(* CODESYS project mobject-graph-vision-pack.library
   Company: mobject
   Version: 0.7.0
   DefaultNamespace: mobject-graph-vision-pack
   Title: mobject-graph-vision-pack
   Placeholder: mobject-graph-vision-pack
   Author: mobject dev team
   DocFormat: reStructuredText

Project tree, tasks and I/O mapping:
  libraries: mobject-core, 0.5.0 (mobject); mobject-graph, 0.14.0 (mobject); mobject-graph-plc-pack, 0.15.0 (mobject); Tc2_Standard, * (Beckhoff Automation GmbH); Tc2_System, * (Beckhoff Automation GmbH); Tc3_Module, * (Beckhoff Automation GmbH); Tc3_Vision, * (Beckhoff Automation GmbH)
  Datatypes/
    Aliases/
      function block _GVCP_REGISTER_ADDRESS [ST]: SetBaseDatatypeReference, Address, ClearReference, Size, FB_init, Clone, Identifier, MakeReferenceTo, TryMakeReferenceTo, Value
      function block _TcVnArray10_ITcVnImage [ST]: SetBaseDatatypeReference, Address, ClearReference, Size, FB_init, Clone, Identifier, MakeReferenceTo, TryMakeReferenceTo, Value
      function block _TcVnArray3_Point2_REAL [ST]: SetBaseDatatypeReference, Address, ClearReference, Size, FB_init, Clone, Identifier, MakeReferenceTo, TryMakeReferenceTo, Value
      function block _TcVnArray4_LREAL [ST]: SetBaseDatatypeReference, Address, ClearReference, Size, FB_init, Clone, Identifier, MakeReferenceTo, TryMakeReferenceTo, Value
      function block _TcVnArray4_Point2_REAL [ST]: SetBaseDatatypeReference, Address, ClearReference, Size, FB_init, Clone, Identifier, MakeReferenceTo, TryMakeReferenceTo, Value
      function block _TcVnArray7_LREAL [ST]: SetBaseDatatypeReference, Address, ClearReference, Size, FB_init, Clone, Identifier, MakeReferenceTo, TryMakeReferenceTo, Value
      function block _TcVnArray8_LREAL [ST]: SetBaseDatatypeReference, Address, ClearReference, Size, FB_init, Clone, Identifier, MakeReferenceTo, TryMakeReferenceTo, Value
      function block _TcVnPoint [ST]: SetBaseDatatypeReference, Address, ClearReference, Size, FB_init, Clone, Identifier, MakeReferenceTo, TryMakeReferenceTo, Value
      function block _TcVnPoint2_DINT [ST]: SetBaseDatatypeReference, Address, ClearReference, Size, FB_init, Clone, Identifier, MakeReferenceTo, TryMakeReferenceTo, Value
      function block _TcVnPoint2_LREAL [ST]: SetBaseDatatypeReference, Address, ClearReference, Size, FB_init, Clone, Identifier, MakeReferenceTo, TryMakeReferenceTo, Value
      function block _TcVnPoint2_REAL [ST]: SetBaseDatatypeReference, Address, ClearReference, Size, FB_init, Clone, Identifier, MakeReferenceTo, TryMakeReferenceTo, Value
      function block _TcVnPoint3_LREAL [ST]: SetBaseDatatypeReference, Address, ClearReference, Size, FB_init, Clone, Identifier, MakeReferenceTo, TryMakeReferenceTo, Value
      function block _TcVnPoint3_REAL [ST]: SetBaseDatatypeReference, Address, ClearReference, Size, FB_init, Clone, Identifier, MakeReferenceTo, TryMakeReferenceTo, Value
      function block _TcVnRectangle [ST]: SetBaseDatatypeReference, Address, ClearReference, Size, FB_init, Clone, Identifier, MakeReferenceTo, TryMakeReferenceTo, Value
      function block _TcVnVector2_DINT [ST]: SetBaseDatatypeReference, Address, ClearReference, Size, FB_init, Clone, Identifier, MakeReferenceTo, TryMakeReferenceTo, Value
      function block _TcVnVector2_INT [ST]: SetBaseDatatypeReference, Address, ClearReference, Size, FB_init, Clone, Identifier, MakeReferenceTo, TryMakeReferenceTo, Value
      function block _TcVnVector2_LREAL [ST]: SetBaseDatatypeReference, Address, ClearReference, Size, FB_init, Clone, Identifier, MakeReferenceTo, TryMakeReferenceTo, Value
      function block _TcVnVector2_REAL [ST]: SetBaseDatatypeReference, Address, ClearReference, Size, FB_init, Clone, Identifier, MakeReferenceTo, TryMakeReferenceTo, Value
      function block _TcVnVector2_SINT [ST]: SetBaseDatatypeReference, Address, ClearReference, Size, FB_init, Clone, Identifier, MakeReferenceTo, TryMakeReferenceTo, Value
      function block _TcVnVector2_UINT [ST]: SetBaseDatatypeReference, Address, ClearReference, Size, FB_init, Clone, Identifier, MakeReferenceTo, TryMakeReferenceTo, Value
      function block _TcVnVector2_USINT [ST]: SetBaseDatatypeReference, Address, ClearReference, Size, FB_init, Clone, Identifier, MakeReferenceTo, TryMakeReferenceTo, Value
      function block _TcVnVector3_INT [ST]: SetBaseDatatypeReference, Address, ClearReference, Size, FB_init, Clone, Identifier, MakeReferenceTo, TryMakeReferenceTo, Value
      function block _TcVnVector3_LREAL [ST]: SetBaseDatatypeReference, Address, ClearReference, Size, FB_init, Clone, Identifier, MakeReferenceTo, TryMakeReferenceTo, Value
      function block _TcVnVector3_REAL [ST]: SetBaseDatatypeReference, Address, ClearReference, Size, FB_init, Clone, Identifier, MakeReferenceTo, TryMakeReferenceTo, Value
      function block _TcVnVector3_SINT [ST]: SetBaseDatatypeReference, Address, ClearReference, Size, FB_init, Clone, Identifier, MakeReferenceTo, TryMakeReferenceTo, Value
      function block _TcVnVector3_UINT [ST]: SetBaseDatatypeReference, Address, ClearReference, Size, FB_init, Clone, Identifier, MakeReferenceTo, TryMakeReferenceTo, Value
      function block _TcVnVector3_USINT [ST]: SetBaseDatatypeReference, Address, ClearReference, Size, FB_init, Clone, Identifier, MakeReferenceTo, TryMakeReferenceTo, Value
      function block _TcVnVector4_DINT [ST]: SetBaseDatatypeReference, Address, ClearReference, Size, FB_init, Clone, Identifier, MakeReferenceTo, TryMakeReferenceTo, Value
      function block _TcVnVector4_INT [ST]: SetBaseDatatypeReference, Address, ClearReference, Size, FB_init, Clone, Identifier, MakeReferenceTo, TryMakeReferenceTo, Value
      function block _TcVnVector4_LREAL [ST]: SetBaseDatatypeReference, Address, ClearReference, Size, FB_init, Clone, Identifier, MakeReferenceTo, TryMakeReferenceTo, Value
      function block _TcVnVector4_SINT [ST]: SetBaseDatatypeReference, Address, ClearReference, Size, FB_init, Clone, Identifier, MakeReferenceTo, TryMakeReferenceTo, Value
      function block _TcVnVector4_UINT [ST]: SetBaseDatatypeReference, Address, ClearReference, Size, FB_init, Clone, Identifier, MakeReferenceTo, TryMakeReferenceTo, Value
      function block _TcVnVector4_USINT [ST]: SetBaseDatatypeReference, Address, ClearReference, Size, FB_init, Clone, Identifier, MakeReferenceTo, TryMakeReferenceTo, Value
    Arrays/
      function block _Array0to1_0to2OfLREAL [ST]: FB_init, OnSerializeArrayValues, SetElementReference, TryDeserializeArrayValues, Address, BaseDatatype, ClearReference, Size, TryGetElementAsDatatypeByIndex, TryGetLowerBound, TryGetUpperBound, Clone, MakeReferenceTo, TryMakeReferenceTo, Value
      function block _Array0to1OfDINT [ST]: FB_init, OnSerializeArrayValues, SetElementReference, TryDeserializeArrayValues, Address, BaseDatatype, ClearReference, Size, TryGetElementAsDatatypeByIndex, TryGetLowerBound, TryGetUpperBound, Clone, MakeReferenceTo, TryMakeReferenceTo, Value
      function block _Array0to1OfINT [ST]: FB_init, OnSerializeArrayValues, SetElementReference, TryDeserializeArrayValues, Address, BaseDatatype, ClearReference, Size, TryGetElementAsDatatypeByIndex, TryGetLowerBound, TryGetUpperBound, Clone, MakeReferenceTo, TryMakeReferenceTo, Value
      function block _Array0to1OfLREAL [ST]: FB_init, OnSerializeArrayValues, SetElementReference, TryDeserializeArrayValues, Address, BaseDatatype, ClearReference, Size, TryGetElementAsDatatypeByIndex, TryGetLowerBound, TryGetUpperBound, Clone, MakeReferenceTo, TryMakeReferenceTo, Value
      function block _Array0to1OfREAL [ST]: FB_init, OnSerializeArrayValues, SetElementReference, TryDeserializeArrayValues, Address, BaseDatatype, ClearReference, Size, TryGetElementAsDatatypeByIndex, TryGetLowerBound, TryGetUpperBound, Clone, MakeReferenceTo, TryMakeReferenceTo, Value
      function block _Array0to1OfSINT [ST]: FB_init, OnSerializeArrayValues, SetElementReference, TryDeserializeArrayValues, Address, BaseDatatype, ClearReference, Size, TryGetElementAsDatatypeByIndex, TryGetLowerBound, TryGetUpperBound, Clone, MakeReferenceTo, TryMakeReferenceTo, Value
      function block _Array0to1OfUINT [ST]: FB_init, OnSerializeArrayValues, SetElementReference, TryDeserializeArrayValues, Address, BaseDatatype, ClearReference, Size, TryGetElementAsDatatypeByIndex, TryGetLowerBound, TryGetUpperBound, Clone, MakeReferenceTo, TryMakeReferenceTo, Value
      function block _Array0to1OfUSINT [ST]: FB_init, OnSerializeArrayValues, SetElementReference, TryDeserializeArrayValues, Address, BaseDatatype, ClearReference, Size, TryGetElementAsDatatypeByIndex, TryGetLowerBound, TryGetUpperBound, Clone, MakeReferenceTo, TryMakeReferenceTo, Value
      function block _Array0to2_0to2OfLREAL [ST]: FB_init, OnSerializeArrayValues, SetElementReference, TryDeserializeArrayValues, Address, BaseDatatype, ClearReference, Size, TryGetElementAsDatatypeByIndex, TryGetLowerBound, TryGetUpperBound, Clone, MakeReferenceTo, TryMakeReferenceTo, Value
      function block _Array0to2OfINT [ST]: FB_init, OnSerializeArrayValues, SetElementReference, TryDeserializeArrayValues, Address, BaseDatatype, ClearReference, Size, TryGetElementAsDatatypeByIndex, TryGetLowerBound, TryGetUpperBound, Clone, MakeReferenceTo, TryMakeReferenceTo, Value
      function block _Array0to2OfLREAL [ST]: FB_init, OnSerializeArrayValues, SetElementReference, TryDeserializeArrayValues, Address, BaseDatatype, ClearReference, Size, TryGetElementAsDatatypeByIndex, TryGetLowerBound, TryGetUpperBound, Clone, MakeReferenceTo, TryMakeReferenceTo, Value
      function block _Array0to2OfREAL [ST]: FB_init, OnSerializeArrayValues, SetElementReference, TryDeserializeArrayValues, Address, BaseDatatype, ClearReference, Size, TryGetElementAsDatatypeByIndex, TryGetLowerBound, TryGetUpperBound, Clone, MakeReferenceTo, TryMakeReferenceTo, Value
      function block _Array0to2OfSINT [ST]: FB_init, OnSerializeArrayValues, SetElementReference, TryDeserializeArrayValues, Address, BaseDatatype, ClearReference, Size, TryGetElementAsDatatypeByIndex, TryGetLowerBound, TryGetUpperBound, Clone, MakeReferenceTo, TryMakeReferenceTo, Value
      function block _Array0to2OfTcVnPoint2_REAL [ST]: FB_init, OnSerializeArrayValues, SetElementReference, TryDeserializeArrayValues, Address, BaseDatatype, ClearReference, Size, TryGetElementAsDatatypeByIndex, TryGetLowerBound, TryGetUpperBound, Clone, MakeReferenceTo, TryMakeReferenceTo, Value
      function block _Array0to2OfUINT [ST]: FB_init, OnSerializeArrayValues, SetElementReference, TryDeserializeArrayValues, Address, BaseDatatype, ClearReference, Size, TryGetElementAsDatatypeByIndex, TryGetLowerBound, TryGetUpperBound, Clone, MakeReferenceTo, TryMakeReferenceTo, Value
      function block _Array0to2OfUSINT [ST]: FB_init, OnSerializeArrayValues, SetElementReference, TryDeserializeArrayValues, Address, BaseDatatype, ClearReference, Size, TryGetElementAsDatatypeByIndex, TryGetLowerBound, TryGetUpperBound, Clone, MakeReferenceTo, TryMakeReferenceTo, Value
      function block _Array0to32OfUDINT [ST]: FB_init, OnSerializeArrayValues, SetElementReference, TryDeserializeArrayValues, Address, BaseDatatype, ClearReference, Size, TryGetElementAsDatatypeByIndex, TryGetLowerBound, TryGetUpperBound, Clone, MakeReferenceTo, TryMakeReferenceTo, Value
      function block _Array0to3OfDINT [ST]: FB_init, OnSerializeArrayValues, SetElementReference, TryDeserializeArrayValues, Address, BaseDatatype, ClearReference, Size, TryGetElementAsDatatypeByIndex, TryGetLowerBound, TryGetUpperBound, Clone, MakeReferenceTo, TryMakeReferenceTo, Value
      function block _Array0to3OfINT [ST]: FB_init, OnSerializeArrayValues, SetElementReference, TryDeserializeArrayValues, Address, BaseDatatype, ClearReference, Size, TryGetElementAsDatatypeByIndex, TryGetLowerBound, TryGetUpperBound, Clone, MakeReferenceTo, TryMakeReferenceTo, Value
      function block _Array0to3OfLREAL [ST]: FB_init, OnSerializeArrayValues, SetElementReference, TryDeserializeArrayValues, Address, BaseDatatype, ClearReference, Size, TryGetElementAsDatatypeByIndex, TryGetLowerBound, TryGetUpperBound, Clone, MakeReferenceTo, TryMakeReferenceTo, Value
      function block _Array0to3OfSINT [ST]: FB_init, OnSerializeArrayValues, SetElementReference, TryDeserializeArrayValues, Address, BaseDatatype, ClearReference, Size, TryGetElementAsDatatypeByIndex, TryGetLowerBound, TryGetUpperBound, Clone, MakeReferenceTo, TryMakeReferenceTo, Value
      function block _Array0to3OfTcVnPoint2_REAL [ST]: FB_init, OnSerializeArrayValues, SetElementReference, TryDeserializeArrayValues, Address, BaseDatatype, ClearReference, Size, TryGetElementAsDatatypeByIndex, TryGetLowerBound, TryGetUpperBound, Clone, MakeReferenceTo, TryMakeReferenceTo, Value
      function block _Array0to3OfUINT [ST]: FB_init, OnSerializeArrayValues, SetElementReference, TryDeserializeArrayValues, Address, BaseDatatype, ClearReference, Size, TryGetElementAsDatatypeByIndex, TryGetLowerBound, TryGetUpperBound, Clone, MakeReferenceTo, TryMakeReferenceTo, Value
      function block _Array0to3OfUSINT [ST]: FB_init, OnSerializeArrayValues, SetElementReference, TryDeserializeArrayValues, Address, BaseDatatype, ClearReference, Size, TryGetElementAsDatatypeByIndex, TryGetLowerBound, TryGetUpperBound, Clone, MakeReferenceTo, TryMakeReferenceTo, Value
      function block _Array0to6OfLREAL [ST]: FB_init, OnSerializeArrayValues, SetElementReference, TryDeserializeArrayValues, Address, BaseDatatype, ClearReference, Size, TryGetElementAsDatatypeByIndex, TryGetLowerBound, TryGetUpperBound, Clone, MakeReferenceTo, TryMakeReferenceTo, Value
      function block _Array0to7OfLREAL [ST]: FB_init, OnSerializeArrayValues, SetElementReference, TryDeserializeArrayValues, Address, BaseDatatype, ClearReference, Size, TryGetElementAsDatatypeByIndex, TryGetLowerBound, TryGetUpperBound, Clone, MakeReferenceTo, TryMakeReferenceTo, Value
      function block _Array0to9OfITcVnImage [ST]: FB_init, OnSerializeArrayValues, SetElementReference, TryDeserializeArrayValues, Address, BaseDatatype, ClearReference, Size, TryGetElementAsDatatypeByIndex, TryGetLowerBound, TryGetUpperBound, Clone, MakeReferenceTo, TryMakeReferenceTo, Value
    Enums/
      function block _ETcVn2dCodeSearchStrategy [ST]: SetBaseDatatypeReference, Address, ClearReference, Size, FB_init, AddLocalEnumeration, IsEnumeratorValueEqual, Clone, Identifier, MakeReferenceTo, TryMakeReferenceTo, Value
      function block _ETcVnAdaptiveThresholdMethod [ST]: SetBaseDatatypeReference, Address, ClearReference, Size, FB_init, AddLocalEnumeration, IsEnumeratorValueEqual, Clone, Identifier, MakeReferenceTo, TryMakeReferenceTo, Value
      function block _ETcVnBarcodeSearchDirection [ST]: SetBaseDatatypeReference, Address, ClearReference, Size, FB_init, AddLocalEnumeration, IsEnumeratorValueEqual, Clone, Identifier, MakeReferenceTo, TryMakeReferenceTo, Value
      function block _ETcVnBarcodeType [ST]: SetBaseDatatypeReference, Address, ClearReference, Size, FB_init, AddLocalEnumeration, IsEnumeratorValueEqual, Clone, Identifier, MakeReferenceTo, TryMakeReferenceTo, Value
      function block _ETcVnBlobCombination [ST]: SetBaseDatatypeReference, Address, ClearReference, Size, FB_init, AddLocalEnumeration, IsEnumeratorValueEqual, Clone, Identifier, MakeReferenceTo, TryMakeReferenceTo, Value
      function block _ETcVnBorderInterpolationMethod [ST]: SetBaseDatatypeReference, Address, ClearReference, Size, FB_init, AddLocalEnumeration, IsEnumeratorValueEqual, Clone, Identifier, MakeReferenceTo, TryMakeReferenceTo, Value
      function block _ETcVnCalibrationPattern [ST]: SetBaseDatatypeReference, Address, ClearReference, Size, FB_init, AddLocalEnumeration, IsEnumeratorValueEqual, Clone, Identifier, MakeReferenceTo, TryMakeReferenceTo, Value
      function block _ETcVnCalibrationPatternOrigin [ST]: SetBaseDatatypeReference, Address, ClearReference, Size, FB_init, AddLocalEnumeration, IsEnumeratorValueEqual, Clone, Identifier, MakeReferenceTo, TryMakeReferenceTo, Value
      function block _ETcVnCameraState [ST]: SetBaseDatatypeReference, Address, ClearReference, Size, FB_init, AddLocalEnumeration, IsEnumeratorValueEqual, Clone, Identifier, MakeReferenceTo, TryMakeReferenceTo, Value
      function block _ETcVnClusteringAlgorithm [ST]: SetBaseDatatypeReference, Address, ClearReference, Size, FB_init, AddLocalEnumeration, IsEnumeratorValueEqual, Clone, Identifier, MakeReferenceTo, TryMakeReferenceTo, Value
      function block _ETcVnColorMap [ST]: SetBaseDatatypeReference, Address, ClearReference, Size, FB_init, AddLocalEnumeration, IsEnumeratorValueEqual, Clone, Identifier, MakeReferenceTo, TryMakeReferenceTo, Value
      function block _ETcVnColorMapSize [ST]: SetBaseDatatypeReference, Address, ClearReference, Size, FB_init, AddLocalEnumeration, IsEnumeratorValueEqual, Clone, Identifier, MakeReferenceTo, TryMakeReferenceTo, Value
      function block _ETcVnColorSpaceTransform [ST]: SetBaseDatatypeReference, Address, ClearReference, Size, FB_init, AddLocalEnumeration, IsEnumeratorValueEqual, Clone, Identifier, MakeReferenceTo, TryMakeReferenceTo, Value
      function block _ETcVnColorTrainingMethod [ST]: SetBaseDatatypeReference, Address, ClearReference, Size, FB_init, AddLocalEnumeration, IsEnumeratorValueEqual, Clone, Identifier, MakeReferenceTo, TryMakeReferenceTo, Value
      function block _ETcVnConnectedComponentsAlgorithm [ST]: SetBaseDatatypeReference, Address, ClearReference, Size, FB_init, AddLocalEnumeration, IsEnumeratorValueEqual, Clone, Identifier, MakeReferenceTo, TryMakeReferenceTo, Value
      function block _ETcVnContainerExportFormat [ST]: SetBaseDatatypeReference, Address, ClearReference, Size, FB_init, AddLocalEnumeration, IsEnumeratorValueEqual, Clone, Identifier, MakeReferenceTo, TryMakeReferenceTo, Value
      function block _ETcVnContourApproximationMethod [ST]: SetBaseDatatypeReference, Address, ClearReference, Size, FB_init, AddLocalEnumeration, IsEnumeratorValueEqual, Clone, Identifier, MakeReferenceTo, TryMakeReferenceTo, Value
      function block _ETcVnContourRetrievalMode [ST]: SetBaseDatatypeReference, Address, ClearReference, Size, FB_init, AddLocalEnumeration, IsEnumeratorValueEqual, Clone, Identifier, MakeReferenceTo, TryMakeReferenceTo, Value
      function block _ETcVnContoursMatchComparisonMethod [ST]: SetBaseDatatypeReference, Address, ClearReference, Size, FB_init, AddLocalEnumeration, IsEnumeratorValueEqual, Clone, Identifier, MakeReferenceTo, TryMakeReferenceTo, Value
      function block _ETcVnDiffusivityTypeKAZE [ST]: SetBaseDatatypeReference, Address, ClearReference, Size, FB_init, AddLocalEnumeration, IsEnumeratorValueEqual, Clone, Identifier, MakeReferenceTo, TryMakeReferenceTo, Value
      function block _ETcVnDistanceTransformationLabel [ST]: SetBaseDatatypeReference, Address, ClearReference, Size, FB_init, AddLocalEnumeration, IsEnumeratorValueEqual, Clone, Identifier, MakeReferenceTo, TryMakeReferenceTo, Value
      function block _ETcVnDistanceTransformationMask [ST]: SetBaseDatatypeReference, Address, ClearReference, Size, FB_init, AddLocalEnumeration, IsEnumeratorValueEqual, Clone, Identifier, MakeReferenceTo, TryMakeReferenceTo, Value
      function block _ETcVnDistanceType [ST]: SetBaseDatatypeReference, Address, ClearReference, Size, FB_init, AddLocalEnumeration, IsEnumeratorValueEqual, Clone, Identifier, MakeReferenceTo, TryMakeReferenceTo, Value
      function block _ETcVnDrawMatchesFlags [ST]: SetBaseDatatypeReference, Address, ClearReference, Size, FB_init, AddLocalEnumeration, IsEnumeratorValueEqual, Clone, Identifier, MakeReferenceTo, TryMakeReferenceTo, Value
      function block _ETcVnDrawShape [ST]: SetBaseDatatypeReference, Address, ClearReference, Size, FB_init, AddLocalEnumeration, IsEnumeratorValueEqual, Clone, Identifier, MakeReferenceTo, TryMakeReferenceTo, Value
      function block _ETcVnEdgeDetectionAlgorithm [ST]: SetBaseDatatypeReference, Address, ClearReference, Size, FB_init, AddLocalEnumeration, IsEnumeratorValueEqual, Clone, Identifier, MakeReferenceTo, TryMakeReferenceTo, Value
      function block _ETcVnEdgeDirection [ST]: SetBaseDatatypeReference, Address, ClearReference, Size, FB_init, AddLocalEnumeration, IsEnumeratorValueEqual, Clone, Identifier, MakeReferenceTo, TryMakeReferenceTo, Value
      function block _ETcVnElementType [ST]: SetBaseDatatypeReference, Address, ClearReference, Size, FB_init, AddLocalEnumeration, IsEnumeratorValueEqual, Clone, Identifier, MakeReferenceTo, TryMakeReferenceTo, Value
      function block _ETcVnEstimationAlgorithm [ST]: SetBaseDatatypeReference, Address, ClearReference, Size, FB_init, AddLocalEnumeration, IsEnumeratorValueEqual, Clone, Identifier, MakeReferenceTo, TryMakeReferenceTo, Value
      function block _ETcVnExtremePointDirection [ST]: SetBaseDatatypeReference, Address, ClearReference, Size, FB_init, AddLocalEnumeration, IsEnumeratorValueEqual, Clone, Identifier, MakeReferenceTo, TryMakeReferenceTo, Value
      function block _ETcVnFeatureDescriptorTypeAKAZE [ST]: SetBaseDatatypeReference, Address, ClearReference, Size, FB_init, AddLocalEnumeration, IsEnumeratorValueEqual, Clone, Identifier, MakeReferenceTo, TryMakeReferenceTo, Value
      function block _ETcVnFeatureScoreTypeORB [ST]: SetBaseDatatypeReference, Address, ClearReference, Size, FB_init, AddLocalEnumeration, IsEnumeratorValueEqual, Clone, Identifier, MakeReferenceTo, TryMakeReferenceTo, Value
      function block _ETcVnFilterDirection [ST]: SetBaseDatatypeReference, Address, ClearReference, Size, FB_init, AddLocalEnumeration, IsEnumeratorValueEqual, Clone, Identifier, MakeReferenceTo, TryMakeReferenceTo, Value
      function block _ETcVnFlipAxis [ST]: SetBaseDatatypeReference, Address, ClearReference, Size, FB_init, AddLocalEnumeration, IsEnumeratorValueEqual, Clone, Identifier, MakeReferenceTo, TryMakeReferenceTo, Value
      function block _ETcVnFontType [ST]: SetBaseDatatypeReference, Address, ClearReference, Size, FB_init, AddLocalEnumeration, IsEnumeratorValueEqual, Clone, Identifier, MakeReferenceTo, TryMakeReferenceTo, Value
      function block _ETcVnHoughMethod [ST]: SetBaseDatatypeReference, Address, ClearReference, Size, FB_init, AddLocalEnumeration, IsEnumeratorValueEqual, Clone, Identifier, MakeReferenceTo, TryMakeReferenceTo, Value
      function block _ETcVnInterpolationType [ST]: SetBaseDatatypeReference, Address, ClearReference, Size, FB_init, AddLocalEnumeration, IsEnumeratorValueEqual, Clone, Identifier, MakeReferenceTo, TryMakeReferenceTo, Value
      function block _ETcVnKeypointDetectionTypeAGAST [ST]: SetBaseDatatypeReference, Address, ClearReference, Size, FB_init, AddLocalEnumeration, IsEnumeratorValueEqual, Clone, Identifier, MakeReferenceTo, TryMakeReferenceTo, Value
      function block _ETcVnKeypointDetectionTypeFAST [ST]: SetBaseDatatypeReference, Address, ClearReference, Size, FB_init, AddLocalEnumeration, IsEnumeratorValueEqual, Clone, Identifier, MakeReferenceTo, TryMakeReferenceTo, Value
      function block _ETcVnLineType [ST]: SetBaseDatatypeReference, Address, ClearReference, Size, FB_init, AddLocalEnumeration, IsEnumeratorValueEqual, Clone, Identifier, MakeReferenceTo, TryMakeReferenceTo, Value
      function block _ETcVnMorphologicalOperator [ST]: SetBaseDatatypeReference, Address, ClearReference, Size, FB_init, AddLocalEnumeration, IsEnumeratorValueEqual, Clone, Identifier, MakeReferenceTo, TryMakeReferenceTo, Value
      function block _ETcVnNormalizationType [ST]: SetBaseDatatypeReference, Address, ClearReference, Size, FB_init, AddLocalEnumeration, IsEnumeratorValueEqual, Clone, Identifier, MakeReferenceTo, TryMakeReferenceTo, Value
      function block _ETcVnOrientationMethod [ST]: SetBaseDatatypeReference, Address, ClearReference, Size, FB_init, AddLocalEnumeration, IsEnumeratorValueEqual, Clone, Identifier, MakeReferenceTo, TryMakeReferenceTo, Value
      function block _ETcVnPixelConnectivity [ST]: SetBaseDatatypeReference, Address, ClearReference, Size, FB_init, AddLocalEnumeration, IsEnumeratorValueEqual, Clone, Identifier, MakeReferenceTo, TryMakeReferenceTo, Value
      function block _ETcVnPixelEncoding [ST]: SetBaseDatatypeReference, Address, ClearReference, Size, FB_init, AddLocalEnumeration, IsEnumeratorValueEqual, Clone, Identifier, MakeReferenceTo, TryMakeReferenceTo, Value
      function block _ETcVnPixelPackMode [ST]: SetBaseDatatypeReference, Address, ClearReference, Size, FB_init, AddLocalEnumeration, IsEnumeratorValueEqual, Clone, Identifier, MakeReferenceTo, TryMakeReferenceTo, Value
      function block _ETcVnRectangleIntersection [ST]: SetBaseDatatypeReference, Address, ClearReference, Size, FB_init, AddLocalEnumeration, IsEnumeratorValueEqual, Clone, Identifier, MakeReferenceTo, TryMakeReferenceTo, Value
      function block _ETcVnRotationAngle [ST]: SetBaseDatatypeReference, Address, ClearReference, Size, FB_init, AddLocalEnumeration, IsEnumeratorValueEqual, Clone, Identifier, MakeReferenceTo, TryMakeReferenceTo, Value
      function block _ETcVnSignedNormalization [ST]: SetBaseDatatypeReference, Address, ClearReference, Size, FB_init, AddLocalEnumeration, IsEnumeratorValueEqual, Clone, Identifier, MakeReferenceTo, TryMakeReferenceTo, Value
      function block _ETcVnStructuringElementShape [ST]: SetBaseDatatypeReference, Address, ClearReference, Size, FB_init, AddLocalEnumeration, IsEnumeratorValueEqual, Clone, Identifier, MakeReferenceTo, TryMakeReferenceTo, Value
      function block _ETcVnTemplateMatchMethod [ST]: SetBaseDatatypeReference, Address, ClearReference, Size, FB_init, AddLocalEnumeration, IsEnumeratorValueEqual, Clone, Identifier, MakeReferenceTo, TryMakeReferenceTo, Value
      function block _ETcVnThresholdType [ST]: SetBaseDatatypeReference, Address, ClearReference, Size, FB_init, AddLocalEnumeration, IsEnumeratorValueEqual, Clone, Identifier, MakeReferenceTo, TryMakeReferenceTo, Value
      function block _ETcVnVectorCompareMethod [ST]: SetBaseDatatypeReference, Address, ClearReference, Size, FB_init, AddLocalEnumeration, IsEnumeratorValueEqual, Clone, Identifier, MakeReferenceTo, TryMakeReferenceTo, Value
      function block _ETcVnWorldCoordinateSystem [ST]: SetBaseDatatypeReference, Address, ClearReference, Size, FB_init, AddLocalEnumeration, IsEnumeratorValueEqual, Clone, Identifier, MakeReferenceTo, TryMakeReferenceTo, Value
      function block _ETcWatchdogAccumulationType [ST]: SetBaseDatatypeReference, Address, ClearReference, Size, FB_init, AddLocalEnumeration, IsEnumeratorValueEqual, Clone, Identifier, MakeReferenceTo, TryMakeReferenceTo, Value
      function block _GEV_CAMERA_STATE [ST]: SetBaseDatatypeReference, Address, ClearReference, Size, FB_init, AddLocalEnumeration, IsEnumeratorValueEqual, Clone, Identifier, MakeReferenceTo, TryMakeReferenceTo, Value
    Interfaces/
      function block _ITcVnContainer [ST]: Address, ClearReference, Size, FB_exit, Serialize_ContainerType_Vector_DINT, Serialize_ContainerType_Vector_INT, Serialize_ContainerType_Vector_ITcVnImage, Serialize_ContainerType_Vector_LREAL, Serialize_ContainerType_Vector_REAL, Serialize_ContainerType_Vector_SINT, Serialize_ContainerType_Vector_UDINT, Serialize_ContainerType_Vector_UINT, Serialize_ContainerType_Vector_ULINT, Serialize_ContainerType_Vector_USINT, TryTcReleaseLocal, Clone, Identifier, MakeReferenceTo, SerializeWith, TryDeserializeFrom, TryMakeReferenceTo, Value, HasType, IsValid, TryGetTypeName, TryTcAddRef, TryTcRelease
      function block _ITcVnImage [ST]: Address, ClearReference, Size, FB_exit, TryGetElementTypeFromInfo, TryTcReleaseLocal, Clone, Identifier, MakeReferenceTo, SerializeWith, TryMakeReferenceTo, Value, HasChannelCount, IsPixelValueCompatible, IsValid, TryDeserializeFrom, TryGetHeight, TryGetImageData, TryGetImageInfo, TryGetImageSize, TryGetPixelFormat, TryGetRowPointer, TryGetWidth, TryGetXPadding, TryGetYPadding, TryReleaseRowPointer, TryTcAddRef, TryTcRelease
    Structs/
      function block _TcVnCircularArc [ST]: Address, ClearReference, Size, FB_init, SetMemberReference, Clone, Identifier, MakeReferenceTo, TryMakeReferenceTo, Value, aCenter, fEndAngle, fRadius, fStartAngle
      function block _TcVnDMatch [ST]: Address, ClearReference, Size, FB_init, SetMemberReference, Clone, Identifier, MakeReferenceTo, TryMakeReferenceTo, Value, fDistance, nImageIdx, nQueryIdx, nTrainIdx
      function block _TcVnImageInfo [ST]: Address, ClearReference, Size, FB_init, SetMemberReference, Clone, Identifier, MakeReferenceTo, TryMakeReferenceTo, Value, nHeight, nImageSize, nWidth, nXPadding, nYPadding, stPixelFormat
      function block _TcVnKeyPoint [ST]: Address, ClearReference, Size, FB_init, SetMemberReference, Clone, Identifier, MakeReferenceTo, TryMakeReferenceTo, Value, aPoint, fAngle, fDiameter, fResponse, nClassId, nOctave
      function block _TcVnParamsBlobDetection [ST]: Address, ClearReference, Size, FB_init, SetMemberReference, Clone, Identifier, MakeReferenceTo, TryMakeReferenceTo, Value, bFilterByArea, bFilterByCircularity, bFilterByConvexity, bFilterByEccentricity, bFilterByInertiaRatio, eBlobCombination, eThresholdType, fMaxArea, fMaxCircularity, fMaxConvexity, fMaxEccentricity, fMaxInertiaRatio, fMaxThreshold, fMinArea, fMinBlobDistance, fMinCircularity, fMinConvexity, fMinEccentricity, fMinInertiaRatio, fMinThreshold, fThresholdStep, nMinRepeatability
      function block _TcVnPixelFormat [ST]: Address, ClearReference, Size, FB_init, SetMemberReference, Clone, Identifier, MakeReferenceTo, TryMakeReferenceTo, Value, bFloat, bPlanar, bSigned, bSupported, ePixelEncoding, ePixelPackMode, nChannels, nElementSize, nTotalSize
      function block _TcVnRectangle_DINT [ST]: Address, ClearReference, Size, FB_init, SetMemberReference, Clone, Identifier, MakeReferenceTo, TryMakeReferenceTo, Value, nHeight, nWidth, nX, nY
      function block _TcVnRectangle_UDINT [ST]: Address, ClearReference, Size, FB_init, SetMemberReference, Clone, Identifier, MakeReferenceTo, TryMakeReferenceTo, Value, nHeight, nWidth, nX, nY
      function block _TcVnRotatedRectangle [ST]: Address, ClearReference, Size, FB_init, SetMemberReference, Clone, Identifier, MakeReferenceTo, TryMakeReferenceTo, Value, aCenter, fAngle, stSize
      function block _TcVnSize2_REAL [ST]: Address, ClearReference, Size, FB_init, SetMemberReference, Clone, Identifier, MakeReferenceTo, TryMakeReferenceTo, Value, fHeight, fWidth
    function block VisionDatatypePack [ST]: RegisterWithDatatypes
  Nodes/
    Algebraic Container Operations/
    Algebraic Image Operations/
      function block Node_F_VN_BitwiseAndImages [ST]: FB_init, Clone, OnExecute, PreExecutionCheck
      function block Node_F_VN_BitwiseNotImage [ST]: FB_init, Clone, OnExecute, PreExecutionCheck
      function block Node_F_VN_BitwiseOrImages [ST]: FB_init, Clone, OnExecute, PreExecutionCheck
      function block Node_F_VN_BitwiseXorImages [ST]: FB_init, Clone, OnExecute, PreExecutionCheck
    Basic Container Operations/
      function block Node_F_VN_AppendToContainer_DINT [ST]: FB_init, Clone, OnExecute, PreExecutionCheck
      function block Node_F_VN_AppendToContainer_INT [ST]: FB_init, Clone, OnExecute, PreExecutionCheck
      function block Node_F_VN_AppendToContainer_ITcVnContainer [ST]: FB_init, Clone, OnExecute, PreExecutionCheck
      function block Node_F_VN_AppendToContainer_ITcVnImage [ST]: FB_init, Clone, OnExecute, PreExecutionCheck
      function block Node_F_VN_AppendToContainer_LREAL [ST]: FB_init, Clone, OnExecute, PreExecutionCheck
      function block Node_F_VN_AppendToContainer_REAL [ST]: FB_init, Clone, OnExecute, PreExecutionCheck
      function block Node_F_VN_AppendToContainer_SINT [ST]: FB_init, Clone, OnExecute, PreExecutionCheck
      function block Node_F_VN_AppendToContainer_TcVnDMatch [ST]: FB_init, Clone, OnExecute, PreExecutionCheck
      function block Node_F_VN_AppendToContainer_TcVnKeyPoint [ST]: FB_init, Clone, OnExecute, PreExecutionCheck
      function block Node_F_VN_AppendToContainer_TcVnPoint2_DINT [ST]: FB_init, Clone, OnExecute, PreExecutionCheck
      function block Node_F_VN_AppendToContainer_TcVnPoint2_LREAL [ST]: FB_init, Clone, OnExecute, PreExecutionCheck
      function block Node_F_VN_AppendToContainer_TcVnPoint2_REAL [ST]: FB_init, Clone, OnExecute, PreExecutionCheck
      function block Node_F_VN_AppendToContainer_TcVnPoint3_LREAL [ST]: FB_init, Clone, OnExecute, PreExecutionCheck
      function block Node_F_VN_AppendToContainer_TcVnPoint3_REAL [ST]: FB_init, Clone, OnExecute, PreExecutionCheck
      function block Node_F_VN_AppendToContainer_TcVnRectangle_DINT [ST]: FB_init, Clone, OnExecute, PreExecutionCheck
      function block Node_F_VN_AppendToContainer_TcVnVector2_DINT [ST]: FB_init, Clone, OnExecute, PreExecutionCheck
      function block Node_F_VN_AppendToContainer_TcVnVector2_INT [ST]: FB_init, Clone, OnExecute, PreExecutionCheck
      function block Node_F_VN_AppendToContainer_TcVnVector2_REAL [ST]: FB_init, Clone, OnExecute, PreExecutionCheck
      function block Node_F_VN_AppendToContainer_TcVnVector2_SINT [ST]: FB_init, Clone, OnExecute, PreExecutionCheck
      function block Node_F_VN_AppendToContainer_TcVnVector2_UINT [ST]: FB_init, Clone, OnExecute, PreExecutionCheck
      function block Node_F_VN_AppendToContainer_TcVnVector2_USINT [ST]: FB_init, Clone, OnExecute, PreExecutionCheck
      function block Node_F_VN_AppendToContainer_TcVnVector3_INT [ST]: FB_init, Clone, OnExecute, PreExecutionCheck
      function block Node_F_VN_AppendToContainer_TcVnVector3_REAL [ST]: FB_init, Clone, OnExecute, PreExecutionCheck
      function block Node_F_VN_AppendToContainer_TcVnVector3_SINT [ST]: FB_init, Clone, OnExecute, PreExecutionCheck
      function block Node_F_VN_AppendToContainer_TcVnVector3_UINT [ST]: FB_init, Clone, OnExecute, PreExecutionCheck
      function block Node_F_VN_AppendToContainer_TcVnVector3_USINT [ST]: FB_init, Clone, OnExecute, PreExecutionCheck
      function block Node_F_VN_AppendToContainer_TcVnVector4_DINT [ST]: FB_init, Clone, OnExecute, PreExecutionCheck
      function block Node_F_VN_AppendToContainer_TcVnVector4_INT [ST]: FB_init, Clone, OnExecute, PreExecutionCheck
      function block Node_F_VN_AppendToContainer_TcVnVector4_LREAL [ST]: FB_init, Clone, OnExecute, PreExecutionCheck
      function block Node_F_VN_AppendToContainer_TcVnVector4_SINT [ST]: FB_init, Clone, OnExecute, PreExecutionCheck
      function block Node_F_VN_AppendToContainer_TcVnVector4_UINT [ST]: FB_init, Clone, OnExecute, PreExecutionCheck
      function block Node_F_VN_AppendToContainer_TcVnVector4_USINT [ST]: FB_init, Clone, OnExecute, PreExecutionCheck
      function block Node_F_VN_AppendToContainer_UDINT [ST]: FB_init, Clone, OnExecute, PreExecutionCheck
      function block Node_F_VN_AppendToContainer_UINT [ST]: FB_init, Clone, OnExecute, PreExecutionCheck
      function block Node_F_VN_AppendToContainer_ULINT [ST]: FB_init, Clone, OnExecute, PreExecutionCheck
      function block Node_F_VN_AppendToContainer_USINT [ST]: FB_init, Clone, OnExecute, PreExecutionCheck
      function block Node_F_VN_FillContainer_DINT [ST]: FB_init, Clone, OnExecute, PreExecutionCheck
      function block Node_F_VN_FillContainer_INT [ST]: FB_init, Clone, OnExecute, PreExecutionCheck
      function block Node_F_VN_FillContainer_ITcVnImage [ST]: FB_init, Clone, OnExecute, PreExecutionCheck
      function block Node_F_VN_FillContainer_LREAL [ST]: FB_init, Clone, OnExecute, PreExecutionCheck
      function block Node_F_VN_FillContainer_REAL [ST]: FB_init, Clone, OnExecute, PreExecutionCheck
      function block Node_F_VN_FillContainer_SINT [ST]: FB_init, Clone, OnExecute, PreExecutionCheck
      function block Node_F_VN_FillContainer_TcVnDMatch [ST]: FB_init, Clone, OnExecute, PreExecutionCheck
      function block Node_F_VN_FillContainer_TcVnKeyPoint [ST]: FB_init, Clone, OnExecute, PreExecutionCheck
      function block Node_F_VN_FillContainer_TcVnPoint2_DINT [ST]: FB_init, Clone, OnExecute, PreExecutionCheck
      function block Node_F_VN_FillContainer_TcVnPoint2_LREAL [ST]: FB_init, Clone, OnExecute, PreExecutionCheck
      function block Node_F_VN_FillContainer_TcVnPoint2_REAL [ST]: FB_init, Clone, OnExecute, PreExecutionCheck
      function block Node_F_VN_FillContainer_TcVnPoint3_LREAL [ST]: FB_init, Clone, OnExecute, PreExecutionCheck
      function block Node_F_VN_FillContainer_TcVnPoint3_REAL [ST]: FB_init, Clone, OnExecute, PreExecutionCheck
      function block Node_F_VN_FillContainer_TcVnRectangle_DINT [ST]: FB_init, Clone, OnExecute, PreExecutionCheck
      function block Node_F_VN_FillContainer_TcVnVector2_DINT [ST]: FB_init, Clone, OnExecute, PreExecutionCheck
      function block Node_F_VN_FillContainer_TcVnVector2_INT [ST]: FB_init, Clone, OnExecute, PreExecutionCheck
      function block Node_F_VN_FillContainer_TcVnVector2_REAL [ST]: FB_init, Clone, OnExecute, PreExecutionCheck
      function block Node_F_VN_FillContainer_TcVnVector2_SINT [ST]: FB_init, Clone, OnExecute, PreExecutionCheck
      function block Node_F_VN_FillContainer_TcVnVector2_UINT [ST]: FB_init, Clone, OnExecute, PreExecutionCheck
      function block Node_F_VN_FillContainer_TcVnVector2_USINT [ST]: FB_init, Clone, OnExecute, PreExecutionCheck
      function block Node_F_VN_FillContainer_TcVnVector3_INT [ST]: FB_init, Clone, OnExecute, PreExecutionCheck
      function block Node_F_VN_FillContainer_TcVnVector3_REAL [ST]: FB_init, Clone, OnExecute, PreExecutionCheck
      function block Node_F_VN_FillContainer_TcVnVector3_SINT [ST]: FB_init, Clone, OnExecute, PreExecutionCheck
      function block Node_F_VN_FillContainer_TcVnVector3_UINT [ST]: FB_init, Clone, OnExecute, PreExecutionCheck
      function block Node_F_VN_FillContainer_TcVnVector3_USINT [ST]: FB_init, Clone, OnExecute, PreExecutionCheck
      function block Node_F_VN_FillContainer_TcVnVector4_DINT [ST]: FB_init, Clone, OnExecute, PreExecutionCheck
      function block Node_F_VN_FillContainer_TcVnVector4_INT [ST]: FB_init, Clone, OnExecute, PreExecutionCheck
      function block Node_F_VN_FillContainer_TcVnVector4_LREAL [ST]: FB_init, Clone, OnExecute, PreExecutionCheck
      function block Node_F_VN_FillContainer_TcVnVector4_SINT [ST]: FB_init, Clone, OnExecute, PreExecutionCheck
      function block Node_F_VN_FillContainer_TcVnVector4_UINT [ST]: FB_init, Clone, OnExecute, PreExecutionCheck
      function block Node_F_VN_FillContainer_TcVnVector4_USINT [ST]: FB_init, Clone, OnExecute, PreExecutionCheck
      function block Node_F_VN_FillContainer_UDINT [ST]: FB_init, Clone, OnExecute, PreExecutionCheck
      function block Node_F_VN_FillContainer_UINT [ST]: FB_init, Clone, OnExecute, PreExecutionCheck
      function block Node_F_VN_FillContainer_ULINT [ST]: FB_init, Clone, OnExecute, PreExecutionCheck
      function block Node_F_VN_FillContainer_USINT [ST]: FB_init, Clone, OnExecute, PreExecutionCheck
      function block Node_F_VN_GetNumberOfElements [ST]: FB_init, Clone, OnExecute, PreExecutionCheck
      function block Node_F_VN_InsertIntoContainer_DINT [ST]: FB_init, Clone, OnExecute, PreExecutionCheck
      function block Node_F_VN_InsertIntoContainer_INT [ST]: FB_init, Clone, OnExecute, PreExecutionCheck
      function block Node_F_VN_InsertIntoContainer_ITcVnContainer [ST]: FB_init, Clone, OnExecute, PreExecutionCheck
      function block Node_F_VN_InsertIntoContainer_ITcVnImage [ST]: FB_init, Clone, OnExecute, PreExecutionCheck
      function block Node_F_VN_InsertIntoContainer_LREAL [ST]: FB_init, Clone, OnExecute, PreExecutionCheck
      function block Node_F_VN_InsertIntoContainer_REAL [ST]: FB_init, Clone, OnExecute, PreExecutionCheck
      function block Node_F_VN_InsertIntoContainer_SINT [ST]: FB_init, Clone, OnExecute, PreExecutionCheck
      function block Node_F_VN_InsertIntoContainer_TcVnDMatch [ST]: FB_init, Clone, OnExecute, PreExecutionCheck
      function block Node_F_VN_InsertIntoContainer_TcVnKeyPoint [ST]: FB_init, Clone, OnExecute, PreExecutionCheck
      function block Node_F_VN_InsertIntoContainer_TcVnPoint2_DINT [ST]: FB_init, Clone, OnExecute, PreExecutionCheck
      function block Node_F_VN_InsertIntoContainer_TcVnPoint2_LREAL [ST]: FB_init, Clone, OnExecute, PreExecutionCheck
      function block Node_F_VN_InsertIntoContainer_TcVnPoint2_REAL [ST]: FB_init, Clone, OnExecute, PreExecutionCheck
      function block Node_F_VN_InsertIntoContainer_TcVnPoint3_LREAL [ST]: FB_init, Clone, OnExecute, PreExecutionCheck
      function block Node_F_VN_InsertIntoContainer_TcVnPoint3_REAL [ST]: FB_init, Clone, OnExecute, PreExecutionCheck
      function block Node_F_VN_InsertIntoContainer_TcVnRectangle_DINT [ST]: FB_init, Clone, OnExecute, PreExecutionCheck
      function block Node_F_VN_InsertIntoContainer_TcVnVector2_DINT [ST]: FB_init, Clone, OnExecute, PreExecutionCheck
      function block Node_F_VN_InsertIntoContainer_TcVnVector2_INT [ST]: FB_init, Clone, OnExecute, PreExecutionCheck
      function block Node_F_VN_InsertIntoContainer_TcVnVector2_REAL [ST]: FB_init, Clone, OnExecute, PreExecutionCheck
      function block Node_F_VN_InsertIntoContainer_TcVnVector2_SINT [ST]: FB_init, Clone, OnExecute, PreExecutionCheck
      function block Node_F_VN_InsertIntoContainer_TcVnVector2_UINT [ST]: FB_init, Clone, OnExecute, PreExecutionCheck
      function block Node_F_VN_InsertIntoContainer_TcVnVector2_USINT [ST]: FB_init, Clone, OnExecute, PreExecutionCheck
      function block Node_F_VN_InsertIntoContainer_TcVnVector3_INT [ST]: FB_init, Clone, OnExecute, PreExecutionCheck
      function block Node_F_VN_InsertIntoContainer_TcVnVector3_REAL [ST]: FB_init, Clone, OnExecute, PreExecutionCheck
      function block Node_F_VN_InsertIntoContainer_TcVnVector3_SINT [ST]: FB_init, Clone, OnExecute, PreExecutionCheck
      function block Node_F_VN_InsertIntoContainer_TcVnVector3_UINT [ST]: FB_init, Clone, OnExecute, PreExecutionCheck
      function block Node_F_VN_InsertIntoContainer_TcVnVector3_USINT [ST]: FB_init, Clone, OnExecute, PreExecutionCheck
      function block Node_F_VN_InsertIntoContainer_TcVnVector4_DINT [ST]: FB_init, Clone, OnExecute, PreExecutionCheck
      function block Node_F_VN_InsertIntoContainer_TcVnVector4_INT [ST]: FB_init, Clone, OnExecute, PreExecutionCheck
      function block Node_F_VN_InsertIntoContainer_TcVnVector4_LREAL [ST]: FB_init, Clone, OnExecute, PreExecutionCheck
      function block Node_F_VN_InsertIntoContainer_TcVnVector4_SINT [ST]: FB_init, Clone, OnExecute, PreExecutionCheck
      function block Node_F_VN_InsertIntoContainer_TcVnVector4_UINT [ST]: FB_init, Clone, OnExecute, PreExecutionCheck
      function block Node_F_VN_InsertIntoContainer_TcVnVector4_USINT [ST]: FB_init, Clone, OnExecute, PreExecutionCheck
      function block Node_F_VN_InsertIntoContainer_UDINT [ST]: FB_init, Clone, OnExecute, PreExecutionCheck
      function block Node_F_VN_InsertIntoContainer_UINT [ST]: FB_init, Clone, OnExecute, PreExecutionCheck
      function block Node_F_VN_InsertIntoContainer_ULINT [ST]: FB_init, Clone, OnExecute, PreExecutionCheck
      function block Node_F_VN_InsertIntoContainer_USINT [ST]: FB_init, Clone, OnExecute, PreExecutionCheck
      function block Node_F_VN_SetAt_DINT [ST]: FB_init, Clone, OnExecute, PreExecutionCheck
      function block Node_F_VN_SetAt_INT [ST]: FB_init, Clone, OnExecute, PreExecutionCheck
      function block Node_F_VN_SetAt_ITcVnContainer [ST]: FB_init, Clone, OnExecute, PreExecutionCheck
      function block Node_F_VN_SetAt_ITcVnImage [ST]: FB_init, Clone, OnExecute, PreExecutionCheck
      function block Node_F_VN_SetAt_LREAL [ST]: FB_init, Clone, OnExecute, PreExecutionCheck
      function block Node_F_VN_SetAt_REAL [ST]: FB_init, Clone, OnExecute, PreExecutionCheck
      function block Node_F_VN_SetAt_SINT [ST]: FB_init, Clone, OnExecute, PreExecutionCheck
      function block Node_F_VN_SetAt_TcVnDMatch [ST]: FB_init, Clone, OnExecute, PreExecutionCheck
      function block Node_F_VN_SetAt_TcVnKeyPoint [ST]: FB_init, Clone, OnExecute, PreExecutionCheck
      function block Node_F_VN_SetAt_TcVnPoint2_DINT [ST]: FB_init, Clone, OnExecute, PreExecutionCheck
      function block Node_F_VN_SetAt_TcVnPoint2_LREAL [ST]: FB_init, Clone, OnExecute, PreExecutionCheck
      function block Node_F_VN_SetAt_TcVnPoint2_REAL [ST]: FB_init, Clone, OnExecute, PreExecutionCheck
      function block Node_F_VN_SetAt_TcVnPoint3_LREAL [ST]: FB_init, Clone, OnExecute, PreExecutionCheck
      function block Node_F_VN_SetAt_TcVnPoint3_REAL [ST]: FB_init, Clone, OnExecute, PreExecutionCheck
      function block Node_F_VN_SetAt_TcVnRectangle_DINT [ST]: FB_init, Clone, OnExecute, PreExecutionCheck
      function block Node_F_VN_SetAt_TcVnVector2_DINT [ST]: FB_init, Clone, OnExecute, PreExecutionCheck
      function block Node_F_VN_SetAt_TcVnVector2_INT [ST]: FB_init, Clone, OnExecute, PreExecutionCheck
      function block Node_F_VN_SetAt_TcVnVector2_REAL [ST]: FB_init, Clone, OnExecute, PreExecutionCheck
      function block Node_F_VN_SetAt_TcVnVector2_SINT [ST]: FB_init, Clone, OnExecute, PreExecutionCheck
      function block Node_F_VN_SetAt_TcVnVector2_UINT [ST]: FB_init, Clone, OnExecute, PreExecutionCheck
      function block Node_F_VN_SetAt_TcVnVector2_USINT [ST]: FB_init, Clone, OnExecute, PreExecutionCheck
      function block Node_F_VN_SetAt_TcVnVector3_INT [ST]: FB_init, Clone, OnExecute, PreExecutionCheck
      function block Node_F_VN_SetAt_TcVnVector3_REAL [ST]: FB_init, Clone, OnExecute, PreExecutionCheck
      function block Node_F_VN_SetAt_TcVnVector3_SINT [ST]: FB_init, Clone, OnExecute, PreExecutionCheck
      function block Node_F_VN_SetAt_TcVnVector3_UINT [ST]: FB_init, Clone, OnExecute, PreExecutionCheck
      function block Node_F_VN_SetAt_TcVnVector3_USINT [ST]: FB_init, Clone, OnExecute, PreExecutionCheck
      function block Node_F_VN_SetAt_TcVnVector4_DINT [ST]: FB_init, Clone, OnExecute, PreExecutionCheck
      function block Node_F_VN_SetAt_TcVnVector4_INT [ST]: FB_init, Clone, OnExecute, PreExecutionCheck
      function block Node_F_VN_SetAt_TcVnVector4_LREAL [ST]: FB_init, Clone, OnExecute, PreExecutionCheck
      function block Node_F_VN_SetAt_TcVnVector4_SINT [ST]: FB_init, Clone, OnExecute, PreExecutionCheck
      function block Node_F_VN_SetAt_TcVnVector4_UINT [ST]: FB_init, Clone, OnExecute, PreExecutionCheck
      function block Node_F_VN_SetAt_TcVnVector4_USINT [ST]: FB_init, Clone, OnExecute, PreExecutionCheck
      function block Node_F_VN_SetAt_UDINT [ST]: FB_init, Clone, OnExecute, PreExecutionCheck
      function block Node_F_VN_SetAt_UINT [ST]: FB_init, Clone, OnExecute, PreExecutionCheck
      function block Node_F_VN_SetAt_ULINT [ST]: FB_init, Clone, OnExecute, PreExecutionCheck
      function block Node_F_VN_SetAt_USINT [ST]: FB_init, Clone, OnExecute, PreExecutionCheck
    Basic Image Operations/
      function block Node_F_VN_CopyImage [ST]: FB_init, Clone, OnExecute, PreExecutionCheck
      function block Node_F_VN_GetImageChannel [ST]: FB_init, Clone, OnExecute, PreExecutionCheck
      function block Node_F_VN_GetImageHeight [ST]: FB_init, Clone, OnExecute, PreExecutionCheck
      function block Node_F_VN_GetImageInfo [ST]: FB_init, Clone, OnExecute, PreExecutionCheck
      function block Node_F_VN_GetImageWidth [ST]: FB_init, Clone, OnExecute, PreExecutionCheck
      function block Node_F_VN_GetPixelFormat [ST]: FB_init, Clone, OnExecute, PreExecutionCheck
      function block Node_F_VN_SetRoi [ST]: FB_init, Clone, OnExecute, PreExecutionCheck
    Code Quality/
    Code Reading/
    Constants/
      function block Node_RGBA_BLACK [ST]: FB_init, Clone, OnExecute, PreExecutionCheck
      function block Node_RGBA_BLUE [ST]: FB_init, Clone, OnExecute, PreExecutionCheck
      function block Node_RGBA_CYAN [ST]: FB_init, Clone, OnExecute, PreExecutionCheck
      function block Node_RGBA_GREEN [ST]: FB_init, Clone, OnExecute, PreExecutionCheck
      function block Node_RGBA_MAGENTA [ST]: FB_init, Clone, OnExecute, PreExecutionCheck
      function block Node_RGBA_RED [ST]: FB_init, Clone, OnExecute, PreExecutionCheck
      function block Node_RGBA_WHITE [ST]: FB_init, Clone, OnExecute, PreExecutionCheck
      function block Node_RGBA_YELLOW [ST]: FB_init, Clone, OnExecute, PreExecutionCheck
    Container Statistics/
      function block Node_F_VN_MaxElementElementwise_DINT [ST]: FB_init, Clone, OnExecute, PreExecutionCheck
      function block Node_F_VN_MaxElementElementwise_INT [ST]: FB_init, Clone, OnExecute, PreExecutionCheck
      function block Node_F_VN_MaxElementElementwise_LREAL [ST]: FB_init, Clone, OnExecute, PreExecutionCheck
      function block Node_F_VN_MaxElementElementwise_REAL [ST]: FB_init, Clone, OnExecute, PreExecutionCheck
      function block Node_F_VN_MaxElementElementwise_SINT [ST]: FB_init, Clone, OnExecute, PreExecutionCheck
      function block Node_F_VN_MaxElementElementwise_TcVnPoint2_DINT [ST]: FB_init, Clone, OnExecute, PreExecutionCheck
      function block Node_F_VN_MaxElementElementwise_TcVnPoint2_LREAL [ST]: FB_init, Clone, OnExecute, PreExecutionCheck
      function block Node_F_VN_MaxElementElementwise_TcVnPoint2_REAL [ST]: FB_init, Clone, OnExecute, PreExecutionCheck
      function block Node_F_VN_MaxElementElementwise_TcVnPoint3_LREAL [ST]: FB_init, Clone, OnExecute, PreExecutionCheck
      function block Node_F_VN_MaxElementElementwise_TcVnPoint3_REAL [ST]: FB_init, Clone, OnExecute, PreExecutionCheck
      function block Node_F_VN_MaxElementElementwise_TcVnVector2_DINT [ST]: FB_init, Clone, OnExecute, PreExecutionCheck
      function block Node_F_VN_MaxElementElementwise_TcVnVector2_INT [ST]: FB_init, Clone, OnExecute, PreExecutionCheck
      function block Node_F_VN_MaxElementElementwise_TcVnVector2_REAL [ST]: FB_init, Clone, OnExecute, PreExecutionCheck
      function block Node_F_VN_MaxElementElementwise_TcVnVector2_SINT [ST]: FB_init, Clone, OnExecute, PreExecutionCheck
      function block Node_F_VN_MaxElementElementwise_TcVnVector2_UINT [ST]: FB_init, Clone, OnExecute, PreExecutionCheck
      function block Node_F_VN_MaxElementElementwise_TcVnVector2_USINT [ST]: FB_init, Clone, OnExecute, PreExecutionCheck
      function block Node_F_VN_MaxElementElementwise_TcVnVector3_INT [ST]: FB_init, Clone, OnExecute, PreExecutionCheck
      function block Node_F_VN_MaxElementElementwise_TcVnVector3_REAL [ST]: FB_init, Clone, OnExecute, PreExecutionCheck
      function block Node_F_VN_MaxElementElementwise_TcVnVector3_SINT [ST]: FB_init, Clone, OnExecute, PreExecutionCheck
      function block Node_F_VN_MaxElementElementwise_TcVnVector3_UINT [ST]: FB_init, Clone, OnExecute, PreExecutionCheck
      function block Node_F_VN_MaxElementElementwise_TcVnVector3_USINT [ST]: FB_init, Clone, OnExecute, PreExecutionCheck
      function block Node_F_VN_MaxElementElementwise_TcVnVector4_DINT [ST]: FB_init, Clone, OnExecute, PreExecutionCheck
      function block Node_F_VN_MaxElementElementwise_TcVnVector4_INT [ST]: FB_init, Clone, OnExecute, PreExecutionCheck
      function block Node_F_VN_MaxElementElementwise_TcVnVector4_LREAL [ST]: FB_init, Clone, OnExecute, PreExecutionCheck
      function block Node_F_VN_MaxElementElementwise_TcVnVector4_SINT [ST]: FB_init, Clone, OnExecute, PreExecutionCheck
      function block Node_F_VN_MaxElementElementwise_TcVnVector4_UINT [ST]: FB_init, Clone, OnExecute, PreExecutionCheck
      function block Node_F_VN_MaxElementElementwise_TcVnVector4_USINT [ST]: FB_init, Clone, OnExecute, PreExecutionCheck
      function block Node_F_VN_MaxElementElementwise_UDINT [ST]: FB_init, Clone, OnExecute, PreExecutionCheck
      function block Node_F_VN_MaxElementElementwise_UINT [ST]: FB_init, Clone, OnExecute, PreExecutionCheck
      function block Node_F_VN_MaxElementElementwise_ULINT [ST]: FB_init, Clone, OnExecute, PreExecutionCheck
      function block Node_F_VN_MaxElementElementwise_USINT [ST]: FB_init, Clone, OnExecute, PreExecutionCheck
      function block Node_F_VN_MedianElementElementwise_DINT [ST]: FB_init, Clone, OnExecute, PreExecutionCheck
      function block Node_F_VN_MedianElementElementwise_INT [ST]: FB_init, Clone, OnExecute, PreExecutionCheck
      function block Node_F_VN_MedianElementElementwise_LREAL [ST]: FB_init, Clone, OnExecute, PreExecutionCheck
      function block Node_F_VN_MedianElementElementwise_REAL [ST]: FB_init, Clone, OnExecute, PreExecutionCheck
      function block Node_F_VN_MedianElementElementwise_SINT [ST]: FB_init, Clone, OnExecute, PreExecutionCheck
      function block Node_F_VN_MedianElementElementwise_TcVnPoint2_DINT [ST]: FB_init, Clone, OnExecute, PreExecutionCheck
      function block Node_F_VN_MedianElementElementwise_TcVnPoint2_LREAL [ST]: FB_init, Clone, OnExecute, PreExecutionCheck
      function block Node_F_VN_MedianElementElementwise_TcVnPoint2_REAL [ST]: FB_init, Clone, OnExecute, PreExecutionCheck
      function block Node_F_VN_MedianElementElementwise_TcVnPoint3_LREAL [ST]: FB_init, Clone, OnExecute, PreExecutionCheck
      function block Node_F_VN_MedianElementElementwise_TcVnPoint3_REAL [ST]: FB_init, Clone, OnExecute, PreExecutionCheck
      function block Node_F_VN_MedianElementElementwise_TcVnVector2_DINT [ST]: FB_init, Clone, OnExecute, PreExecutionCheck
      function block Node_F_VN_MedianElementElementwise_TcVnVector2_INT [ST]: FB_init, Clone, OnExecute, PreExecutionCheck
      function block Node_F_VN_MedianElementElementwise_TcVnVector2_REAL [ST]: FB_init, Clone, OnExecute, PreExecutionCheck
      function block Node_F_VN_MedianElementElementwise_TcVnVector2_SINT [ST]: FB_init, Clone, OnExecute, PreExecutionCheck
      function block Node_F_VN_MedianElementElementwise_TcVnVector2_UINT [ST]: FB_init, Clone, OnExecute, PreExecutionCheck
      function block Node_F_VN_MedianElementElementwise_TcVnVector2_USINT [ST]: FB_init, Clone, OnExecute, PreExecutionCheck
      function block Node_F_VN_MedianElementElementwise_TcVnVector3_INT [ST]: FB_init, Clone, OnExecute, PreExecutionCheck
      function block Node_F_VN_MedianElementElementwise_TcVnVector3_REAL [ST]: FB_init, Clone, OnExecute, PreExecutionCheck
      function block Node_F_VN_MedianElementElementwise_TcVnVector3_SINT [ST]: FB_init, Clone, OnExecute, PreExecutionCheck
      function block Node_F_VN_MedianElementElementwise_TcVnVector3_UINT [ST]: FB_init, Clone, OnExecute, PreExecutionCheck
      function block Node_F_VN_MedianElementElementwise_TcVnVector3_USINT [ST]: FB_init, Clone, OnExecute, PreExecutionCheck
      function block Node_F_VN_MedianElementElementwise_TcVnVector4_DINT [ST]: FB_init, Clone, OnExecute, PreExecutionCheck
      function block Node_F_VN_MedianElementElementwise_TcVnVector4_INT [ST]: FB_init, Clone, OnExecute, PreExecutionCheck
      function block Node_F_VN_MedianElementElementwise_TcVnVector4_LREAL [ST]: FB_init, Clone, OnExecute, PreExecutionCheck
      function block Node_F_VN_MedianElementElementwise_TcVnVector4_SINT [ST]: FB_init, Clone, OnExecute, PreExecutionCheck
      function block Node_F_VN_MedianElementElementwise_TcVnVector4_UINT [ST]: FB_init, Clone, OnExecute, PreExecutionCheck
      function block Node_F_VN_MedianElementElementwise_TcVnVector4_USINT [ST]: FB_init, Clone, OnExecute, PreExecutionCheck
      function block Node_F_VN_MedianElementElementwise_UDINT [ST]: FB_init, Clone, OnExecute, PreExecutionCheck
      function block Node_F_VN_MedianElementElementwise_UINT [ST]: FB_init, Clone, OnExecute, PreExecutionCheck
      function block Node_F_VN_MedianElementElementwise_ULINT [ST]: FB_init, Clone, OnExecute, PreExecutionCheck
      function block Node_F_VN_MedianElementElementwise_USINT [ST]: FB_init, Clone, OnExecute, PreExecutionCheck
      function block Node_F_VN_MinElementElementwise_DINT [ST]: FB_init, Clone, OnExecute, PreExecutionCheck
      function block Node_F_VN_MinElementElementwise_INT [ST]: FB_init, Clone, OnExecute, PreExecutionCheck
      function block Node_F_VN_MinElementElementwise_LREAL [ST]: FB_init, Clone, OnExecute, PreExecutionCheck
      function block Node_F_VN_MinElementElementwise_REAL [ST]: FB_init, Clone, OnExecute, PreExecutionCheck
      function block Node_F_VN_MinElementElementwise_SINT [ST]: FB_init, Clone, OnExecute, PreExecutionCheck
      function block Node_F_VN_MinElementElementwise_TcVnPoint2_DINT [ST]: FB_init, Clone, OnExecute, PreExecutionCheck
      function block Node_F_VN_MinElementElementwise_TcVnPoint2_LREAL [ST]: FB_init, Clone, OnExecute, PreExecutionCheck
      function block Node_F_VN_MinElementElementwise_TcVnPoint2_REAL [ST]: FB_init, Clone, OnExecute, PreExecutionCheck
      function block Node_F_VN_MinElementElementwise_TcVnPoint3_LREAL [ST]: FB_init, Clone, OnExecute, PreExecutionCheck
      function block Node_F_VN_MinElementElementwise_TcVnPoint3_REAL [ST]: FB_init, Clone, OnExecute, PreExecutionCheck
      function block Node_F_VN_MinElementElementwise_TcVnVector2_DINT [ST]: FB_init, Clone, OnExecute, PreExecutionCheck
      function block Node_F_VN_MinElementElementwise_TcVnVector2_INT [ST]: FB_init, Clone, OnExecute, PreExecutionCheck
      function block Node_F_VN_MinElementElementwise_TcVnVector2_REAL [ST]: FB_init, Clone, OnExecute, PreExecutionCheck
      function block Node_F_VN_MinElementElementwise_TcVnVector2_SINT [ST]: FB_init, Clone, OnExecute, PreExecutionCheck
      function block Node_F_VN_MinElementElementwise_TcVnVector2_UINT [ST]: FB_init, Clone, OnExecute, PreExecutionCheck
      function block Node_F_VN_MinElementElementwise_TcVnVector2_USINT [ST]: FB_init, Clone, OnExecute, PreExecutionCheck
      function block Node_F_VN_MinElementElementwise_TcVnVector3_INT [ST]: FB_init, Clone, OnExecute, PreExecutionCheck
      function block Node_F_VN_MinElementElementwise_TcVnVector3_REAL [ST]: FB_init, Clone, OnExecute, PreExecutionCheck
      function block Node_F_VN_MinElementElementwise_TcVnVector3_SINT [ST]: FB_init, Clone, OnExecute, PreExecutionCheck
      function block Node_F_VN_MinElementElementwise_TcVnVector3_UINT [ST]: FB_init, Clone, OnExecute, PreExecutionCheck
      function block Node_F_VN_MinElementElementwise_TcVnVector3_USINT [ST]: FB_init, Clone, OnExecute, PreExecutionCheck
      function block Node_F_VN_MinElementElementwise_TcVnVector4_DINT [ST]: FB_init, Clone, OnExecute, PreExecutionCheck
      function block Node_F_VN_MinElementElementwise_TcVnVector4_INT [ST]: FB_init, Clone, OnExecute, PreExecutionCheck
      function block Node_F_VN_MinElementElementwise_TcVnVector4_LREAL [ST]: FB_init, Clone, OnExecute, PreExecutionCheck
      function block Node_F_VN_MinElementElementwise_TcVnVector4_SINT [ST]: FB_init, Clone, OnExecute, PreExecutionCheck
      function block Node_F_VN_MinElementElementwise_TcVnVector4_UINT [ST]: FB_init, Clone, OnExecute, PreExecutionCheck
      function block Node_F_VN_MinElementElementwise_TcVnVector4_USINT [ST]: FB_init, Clone, OnExecute, PreExecutionCheck
      function block Node_F_VN_MinElementElementwise_UDINT [ST]: FB_init, Clone, OnExecute, PreExecutionCheck
      function block Node_F_VN_MinElementElementwise_UINT [ST]: FB_init, Clone, OnExecute, PreExecutionCheck
      function block Node_F_VN_MinElementElementwise_ULINT [ST]: FB_init, Clone, OnExecute, PreExecutionCheck
      function block Node_F_VN_MinElementElementwise_USINT [ST]: FB_init, Clone, OnExecute, PreExecutionCheck
    Contour Analysis/
      function block Node_F_VN_FitLine [ST]: FB_init, Clone, OnExecute, PreExecutionCheck
    Control Functions/
    Drawing/
      function block Node_F_VN_DrawContours [ST]: FB_init, Clone, OnExecute, PreExecutionCheck
      function block Node_F_VN_DrawLine [ST]: FB_init, Clone, OnExecute, PreExecutionCheck
      function block Node_F_VN_DrawLine_TcVnVector4_LREAL [ST]: FB_init, Clone, OnExecute, PreExecutionCheck
      function block Node_F_VN_PutLabel [ST]: FB_init, Clone, OnExecute, PreExecutionCheck
      function block Node_F_VN_PutText [ST]: FB_init, Clone, OnExecute, PreExecutionCheck
    Fourier Analysis/
    Geometric and Coordinate Transformations/
      function block Node_F_VN_FlipImage [ST]: FB_init, Clone, OnExecute, PreExecutionCheck
    Image Analysis/
      Object Detection/
        function block Node_F_VN_DetectBlobs [ST]: FB_init, Clone, OnExecute, PreExecutionCheck
    Image Color and Contrast Processing/
      function block Node_F_VN_ApplyColorMap [ST]: FB_init, Clone, OnExecute, PreExecutionCheck
      function block Node_F_VN_ConvertColorSpace [ST]: FB_init, Clone, OnExecute, PreExecutionCheck
      function block Node_F_VN_GenerateColorMap [ST]: FB_init, Clone, OnExecute, PreExecutionCheck
    Image Filtering/
      function block Node_F_VN_BoxFilter [ST]: FB_init, Clone, OnExecute, PreExecutionCheck
      function block Node_F_VN_GaussianFilter [ST]: FB_init, Clone, OnExecute, PreExecutionCheck
      function block Node_F_VN_LaplacianFilter [ST]: FB_init, Clone, OnExecute, PreExecutionCheck
    Image Segmentation/
      function block Node_F_VN_Threshold [ST]: FB_init, Clone, OnExecute, PreExecutionCheck
    Keypoint Features/
    Machine Learning/
    Measurement/
      function block Node_F_VN_LocateEdge [ST]: FB_init, Clone, OnExecute, PreExecutionCheck
    Miscellaneous/
    OCR/
    Texture Analysis/
    VisionNode/
      function block VisionNode [ST]: PreExecutionCheck
    function block VisionNodePack [ST]: RegisterWithNodeFactory
  global variables GVL_COLOURS
  function block VisionPack [ST]: RegisterWithDatatypes, RegisterWithNodeFactory
*)

// GVL_COLOURS
{attribute 'qualified_only'}
VAR_GLOBAL
    RGBA_BLACK   : TcVnVector4_LREAL := [0, 0, 0, 255];
    RGBA_RED     : TcVnVector4_LREAL := [255, 0, 0, 255];
    RGBA_YELLOW  : TcVnVector4_LREAL := [255, 255, 0, 255];
    RGBA_GREEN   : TcVnVector4_LREAL := [0, 255, 0, 255];
    RGBA_CYAN    : TcVnVector4_LREAL := [0, 255, 255, 255];
    RGBA_BLUE    : TcVnVector4_LREAL := [0, 0, 255, 255];
    RGBA_MAGENTA : TcVnVector4_LREAL := [255, 0, 255, 255];
    RGBA_WHITE   : TcVnVector4_LREAL := [255, 255, 255, 255];
END_VAR

// Datatypes/Aliases/_GVCP_REGISTER_ADDRESS
{attribute 'linkalways'} 
{attribute 'no_explicit_call' := 'This FB is a CLASS and must be accessed using methods or properties'}
{attribute 'enable_dynamic_creation'}
FUNCTION_BLOCK _GVCP_REGISTER_ADDRESS EXTENDS AliasDatatypeBase
VAR
	localData : GVCP_REGISTER_ADDRESS;
	activeData : REFERENCE TO GVCP_REGISTER_ADDRESS REF= localData;
	aliasBaseDatatype : _UDINT(0);
END_VAR

METHOD PROTECTED SetBaseDatatypeReference
VAR_INPUT
END_VAR
aliasBaseDatatype.MakeReferenceTo(activeData);
END_METHOD

PROPERTY PUBLIC Address : PVOID
GET
Address := ADR(activeData);
END_GET
END_PROPERTY

METHOD PUBLIC ClearReference
VAR_INPUT
END_VAR
activeData REF= localData;
SetBaseDatatypeReference();
END_METHOD

PROPERTY PUBLIC Size : UDINT
GET
Size := SIZEOF(activeData);
END_GET
END_PROPERTY

METHOD FB_init : BOOL
VAR_INPUT
	bInitRetains : BOOL; // if TRUE, the retain variables are initialized (warm start / cold start)
	bInCopyCode : BOOL;  // if TRUE, the instance afterwards gets moved into the copy code (online change)
	//InitialValue : TcVnArray33_UDINT; // if possible, not all values can be initialized
END_VAR
//localData := InitialValue; // if possible, not all values can be initialized
SetBaseDatatypeReference();
AddBaseDatatype(aliasBaseDatatype);
END_METHOD

METHOD PUBLIC Clone : I_Datatype
VAR
    pClone : POINTER TO _GVCP_REGISTER_ADDRESS;
END_VAR
pClone := __NEW(_GVCP_REGISTER_ADDRESS);
Clone := pClone^;
END_METHOD

PROPERTY PUBLIC Identifier : T_MAXSTRING
GET
Identifier := 'GVCP_REGISTER_ADDRESS';
END_GET
END_PROPERTY

METHOD PUBLIC MakeReferenceTo
VAR_INPUT
	ReferenceTarget : REFERENCE TO GVCP_REGISTER_ADDRESS;
END_VAR
activeData REF= ReferenceTarget;
SetBaseDatatypeReference();
END_METHOD

METHOD TryMakeReferenceTo : BOOL
VAR_INPUT
	Target : I_Datatype;
END_VAR
VAR
	pTargetData : POINTER TO GVCP_REGISTER_ADDRESS;
END_VAR
IF NOT IsEquivalentTo(Target) THEN
	RETURN;
END_IF

pTargetData := Target.Address;
activeData REF= pTargetData^;
SetBaseDatatypeReference();
TryMakeReferenceTo := TRUE;
END_METHOD

PROPERTY PUBLIC Value : REFERENCE TO GVCP_REGISTER_ADDRESS
GET
Value REF= activeData;
END_GET
END_PROPERTY

END_FUNCTION_BLOCK

// Datatypes/Aliases/_TcVnArray10_ITcVnImage
{attribute 'linkalways'} 
{attribute 'no_explicit_call' := 'This FB is a CLASS and must be accessed using methods or properties'}
{attribute 'enable_dynamic_creation'}
FUNCTION_BLOCK _TcVnArray10_ITcVnImage EXTENDS AliasDatatypeBase
VAR
	localData : TcVnArray10_ITcVnImage;
	activeData : REFERENCE TO TcVnArray10_ITcVnImage REF= localData;
	aliasBaseDatatype : _Array0to9OfITcVnImage;
END_VAR

METHOD PROTECTED SetBaseDatatypeReference
VAR_INPUT
END_VAR
aliasBaseDatatype.MakeReferenceTo(activeData);
END_METHOD

PROPERTY PUBLIC Address : PVOID
GET
Address := ADR(activeData);
END_GET
END_PROPERTY

METHOD PUBLIC ClearReference
VAR_INPUT
END_VAR
activeData REF= localData;
SetBaseDatatypeReference();
END_METHOD

PROPERTY PUBLIC Size : UDINT
GET
Size := SIZEOF(activeData);
END_GET
END_PROPERTY

METHOD FB_init : BOOL
VAR_INPUT
	bInitRetains : BOOL; // if TRUE, the retain variables are initialized (warm start / cold start)
	bInCopyCode : BOOL;  // if TRUE, the instance afterwards gets moved into the copy code (online change)
	//InitialValue : TcVnArray10_ITcVnImage; // if possible, not all values can be initialized
END_VAR
//localData := InitialValue; // if possible, not all values can be initialized
SetBaseDatatypeReference();
AddBaseDatatype(aliasBaseDatatype);
END_METHOD

METHOD PUBLIC Clone : I_Datatype
VAR
    pClone : POINTER TO _TcVnArray10_ITcVnImage;
END_VAR
pClone := __NEW(_TcVnArray10_ITcVnImage);
Clone := pClone^;
END_METHOD

PROPERTY PUBLIC Identifier : T_MAXSTRING
GET
Identifier := 'TcVnArray10_ITcVnImage';
END_GET
END_PROPERTY

METHOD PUBLIC MakeReferenceTo
VAR_INPUT
	ReferenceTarget : REFERENCE TO TcVnArray10_ITcVnImage;
END_VAR
activeData REF= ReferenceTarget;
SetBaseDatatypeReference();
END_METHOD

METHOD TryMakeReferenceTo : BOOL
VAR_INPUT
	Target : I_Datatype;
END_VAR
VAR
	pTargetData : POINTER TO TcVnArray10_ITcVnImage;
END_VAR
IF NOT IsEquivalentTo(Target) THEN
	RETURN;
END_IF

pTargetData := Target.Address;
activeData REF= pTargetData^;
SetBaseDatatypeReference();
TryMakeReferenceTo := TRUE;
END_METHOD

PROPERTY PUBLIC Value : REFERENCE TO TcVnArray10_ITcVnImage
GET
Value REF= activeData;
END_GET
END_PROPERTY

END_FUNCTION_BLOCK

// Datatypes/Arrays/_Array0to9OfITcVnImage
{attribute 'linkalways'} 
{attribute 'no_explicit_call' := 'This FB is a CLASS and must be accessed using methods or properties'}
{attribute 'enable_dynamic_creation'}
FUNCTION_BLOCK _Array0to9OfITcVnImage EXTENDS ArrayDatatypeBase_1D
VAR CONSTANT
	lBound : DINT := 0;
	uBound : DINT := 9;
END_VAR
VAR
	localData : ARRAY [lBound..uBound] OF ITcVnImage;
	activeData : REFERENCE TO ARRAY [lBound..uBound] OF ITcVnImage REF= localData;
	elements : ARRAY [lBound..uBound] OF _ITcVnImage;
	baseType : _ITcVnImage;
END_VAR

METHOD FB_init : BOOL
VAR_INPUT
	bInitRetains : BOOL; // if TRUE, the retain variables are initialized (warm start / cold start)
	bInCopyCode : BOOL;  // if TRUE, the instance afterwards gets moved into the copy code (online change)
END_VAR
SetElementReference();
END_METHOD

METHOD PROTECTED OnSerializeArrayValues
VAR_INPUT
	Serializer : I_Serializer;
END_VAR
VAR
	i : DINT;
END_VAR
FOR i := lBound TO uBound DO
	elements[i].SerializeWith(Serializer);
END_FOR
END_METHOD

METHOD PROTECTED SetElementReference
VAR_INPUT
END_VAR
VAR
	i : DINT;
END_VAR
FOR i := lBound TO uBound DO
	elements[i].MakeReferenceTo(activeData[i]);
END_FOR
END_METHOD

METHOD PROTECTED TryDeserializeArrayValues : BOOL
VAR_INPUT
	Deserializer : I_Deserializer;
	Feedback : I_DeserializerFeedback;
END_VAR
VAR
	enumerator : I_DeserializerArrayForwardEnumerator;
	i : DINT;
END_VAR
enumerator := Deserializer.GetArrayEnumerator();
i := lBound;

WHILE enumerator.MoveNext() AND i <= uBound DO
	
	IF NOT elements[i].TryDeserializeFrom(enumerator.Current, Feedback) THEN
		EXIT;
	END_IF
	i := i + 1;

END_WHILE
enumerator.Dispose();
END_METHOD

PROPERTY PUBLIC Address : PVOID
GET
Address := ADR(activeData);
END_GET
END_PROPERTY

PROPERTY PUBLIC BaseDatatype : I_Datatype
GET
BaseDatatype := baseType;
END_GET
END_PROPERTY

METHOD PUBLIC ClearReference
VAR_INPUT
END_VAR
activeData REF= localData;
SetElementReference();
END_METHOD

PROPERTY PUBLIC Size : UDINT
GET
Size := SIZEOF(activeData);
END_GET
END_PROPERTY

METHOD PUBLIC TryGetElementAsDatatypeByIndex : BOOL
VAR_INPUT
	Index : DINT;
	Destination : REFERENCE TO I_Datatype;
END_VAR
IF Index < lbound OR Index > ubound THEN
	RETURN;
END_IF

Destination := elements[Index];
TryGetElementAsDatatypeByIndex := TRUE;
END_METHOD

METHOD PUBLIC TryGetLowerBound : BOOL
VAR_INPUT
	Dimention : UDINT;
	Destination : REFERENCE TO DINT;
END_VAR
IF Dimention = 1 THEN
	Destination := lBound;
	TryGetLowerBound := TRUE;
END_IF
END_METHOD

METHOD PUBLIC TryGetUpperBound : BOOL
VAR_INPUT
	Dimention : UDINT;
	Destination : REFERENCE TO DINT;
END_VAR
IF Dimention = 1 THEN
	Destination := uBound;
	TryGetUpperBound := TRUE;
END_IF
END_METHOD

METHOD PUBLIC Clone : I_Datatype
VAR
    pClone : POINTER TO _Array0to9OfITcVnImage;
END_VAR
pClone := __NEW(_Array0to9OfITcVnImage());
pClone^.Value := Value;
Clone := pClone^;
END_METHOD

METHOD PUBLIC MakeReferenceTo
VAR_INPUT
	ReferenceTarget : REFERENCE TO ARRAY [lBound..uBound] OF ITcVnImage;
END_VAR
activeData REF= ReferenceTarget;
SetElementReference();
END_METHOD

METHOD TryMakeReferenceTo : BOOL
VAR_INPUT
	Target : I_Datatype;
END_VAR
VAR
	pTargetData : POINTER TO ARRAY [lBound..uBound] OF ITcVnImage;
END_VAR
IF NOT IsEquivalentTo(Target) THEN
	RETURN;
END_IF

pTargetData := Target.Address;
activeData REF= pTargetData^;
SetElementReference();
TryMakeReferenceTo := TRUE;
END_METHOD

PROPERTY PUBLIC Value : REFERENCE TO ARRAY [lBound..uBound] OF ITcVnImage;
GET
Value ref= activeData;
END_GET
END_PROPERTY

END_FUNCTION_BLOCK

// Datatypes/Interfaces/_ITcVnImage
{attribute 'linkalways'} 
{attribute 'no_explicit_call' := 'This FB is a CLASS and must be accessed using methods or properties'}
{attribute 'enable_dynamic_creation'}
FUNCTION_BLOCK _ITcVnImage EXTENDS InterfaceDatatypeBase
VAR
	localData : ITcVnImage;
	activeData : REFERENCE TO ITcVnImage REF= localData;
END_VAR

PROPERTY PUBLIC Address : PVOID
GET
Address := ADR(activeData);
END_GET
END_PROPERTY

METHOD PUBLIC ClearReference
VAR_INPUT
END_VAR
activeData REF= localData;
END_METHOD

PROPERTY PUBLIC Size : UDINT
GET
Size := SIZEOF(activeData);
END_GET
END_PROPERTY

METHOD FB_exit : BOOL
VAR_INPUT
	bInCopyCode : BOOL; // if TRUE, the exit method is called for exiting an instance that is copied afterwards (online change).
END_VAR
IF bInCopyCode THEN
	RETURN;
END_IF

TryTcReleaseLocal();
END_METHOD

METHOD PRIVATE TryGetElementTypeFromInfo : BOOL;
VAR_INPUT
	ImageInfo : TcVnImageInfo;
	Destination : REFERENCE TO ETcVnElementType;
END_VAR
CASE ImageInfo.stPixelFormat.nElementSize OF
	
	8 : // 8bit
	
		IF ImageInfo.stPixelFormat.bSigned THEN
			Destination := ETcVnElementType.TCVN_ET_SINT;
		ELSE	
			Destination := ETcVnElementType.TCVN_ET_USINT;
		END_IF
		TryGetElementTypeFromInfo := TRUE;
	
	16 : // 16bit
	
		IF ImageInfo.stPixelFormat.bSigned THEN
			Destination := ETcVnElementType.TCVN_ET_INT;
		ELSE	
			Destination := ETcVnElementType.TCVN_ET_UINT;
		END_IF
		TryGetElementTypeFromInfo := TRUE;
	
	32 : // 32bit
	
		IF ImageInfo.stPixelFormat.bSigned AND NOT ImageInfo.stPixelFormat.bFloat THEN
			Destination := ETcVnElementType.TCVN_ET_DINT;
			TryGetElementTypeFromInfo := TRUE;
		END_IF
		
		IF ImageInfo.stPixelFormat.bFloat THEN
			Destination := ETcVnElementType.TCVN_ET_REAL;
			TryGetElementTypeFromInfo := TRUE;
		END_IF
		
	64 : // 64bit
	
		IF ImageInfo.stPixelFormat.bFloat THEN
			Destination := ETcVnElementType.TCVN_ET_LREAL;
			TryGetElementTypeFromInfo := TRUE;
		END_IF
		
ELSE
	
	RETURN;

END_CASE
END_METHOD

METHOD PUBLIC TryTcReleaseLocal : BOOL
VAR_INPUT
END_VAR
IF localData = 0 THEN
	RETURN;
END_IF

IF localData.TcRelease() = 0 THEN
	localData := 0;
END_IF

TryTcReleaseLocal := TRUE;
END_METHOD

METHOD PUBLIC Clone : I_Datatype
VAR
    pClone : POINTER TO _ITcVnImage;
END_VAR
pClone := __NEW(_ITcVnImage);
Clone := pClone^;
END_METHOD

PROPERTY PUBLIC Identifier : T_MAXSTRING
GET
Identifier := 'ITcVnImage';
END_GET
END_PROPERTY

METHOD PUBLIC MakeReferenceTo
VAR_INPUT
	ReferenceTarget : REFERENCE TO ITcVnImage;
END_VAR
activeData REF= ReferenceTarget;
END_METHOD

METHOD PUBLIC SerializeWith
VAR_INPUT
	Serializer : I_Serializer;
END_VAR
VAR
	result: HRESULT;
	exportImageSize: ULINT;
	buffer : POINTER TO BYTE;
	imageInfo : _TcVnImageInfo;
END_VAR
IF NOT (activeData <> 0) THEN
	// no image available, so drop out.. need to add serialization?
	Serializer.AddNull();
	RETURN;
END_IF

result := F_VN_ExportImageSize(ipImage:=activeData, nBufferSize:=exportImageSize, hrPrev:=result);

IF FAILED(result) THEN
	// export to bmp size failed, so drop out.. need to add serialization?
	Serializer.AddNull();
	RETURN;
END_IF

IF exportImageSize > DatatypeLimits.UDINT_MAX_VALUE THEN
	// export is too big for __NEW, so drop out..
	Serializer.AddNull();
	RETURN;
END_IF

IF exportImageSize <= 0 THEN
	// export is zero size, so drop out.. 
	Serializer.AddNull();
	RETURN;
END_IF
	
buffer := __NEW(BYTE,ULINT_TO_UDINT(exportImageSize));
result := F_VN_ExportImage(ipImage:=activeData, pBuffer:=buffer, nBufferSize:=exportImageSize, hrPrev:=result);

IF FAILED(result) THEN
	// export to bmp failed, so drop out.. 
	Serializer.AddNull();
	__DELETE(buffer);
	RETURN;
END_IF

activeData.GetImageInfo(imageInfo.value);

Serializer.StartObject();
Serializer.AddKeyObject('imageInfo',imageInfo);
Serializer.AddKey('imageData');
Serializer.AddBase64(buffer,ULINT_TO_DINT(exportImageSize));
Serializer.EndObject();

__DELETE(buffer);
END_METHOD

METHOD TryMakeReferenceTo : BOOL
VAR_INPUT
	Target : I_Datatype;
END_VAR
VAR
	pTargetData : POINTER TO ITcVnImage;
END_VAR
IF NOT IsEquivalentTo(Target) THEN
	RETURN;
END_IF

pTargetData := Target.Address;
activeData REF= pTargetData^;
TryMakeReferenceTo := TRUE;
END_METHOD

PROPERTY PUBLIC Value : REFERENCE TO ITcVnImage
GET
Value REF= activeData;
END_GET
END_PROPERTY

METHOD PUBLIC HasChannelCount : BOOL
VAR_INPUT
	ChannelCount : BYTE;
END_VAR
VAR
    pixelFormat : TcVnPixelFormat;
END_VAR
IF NOT TryGetPixelFormat(pixelFormat) THEN
    RETURN;
END_IF

IF NOT (pixelFormat.nChannels = ChannelCount) THEN
    RETURN;
END_IF

HasChannelCount := TRUE;
END_METHOD

METHOD PUBLIC IsPixelValueCompatible : BOOL
VAR_INPUT
	PixelValue : LREAL;
END_VAR
END_METHOD

PROPERTY PUBLIC IsValid : BOOL
GET
IsValid := activeData <> 0;
END_GET
END_PROPERTY

METHOD TryDeserializeFrom : BOOL
VAR_INPUT
	Deserializer : I_Deserializer;
	Feedback : I_DeserializerFeedback;
END_VAR
VAR
	imageInfo : _TcVnImageInfo;
	imageSizeInBytes : UDINT;
	buffer : POINTER TO BYTE;
	hr : HRESULT;
	elementType : ETcVnElementType;
END_VAR
IF NOT Deserializer.TryDeserializeKeyToObject('imageInfo', imageInfo, Feedback) THEN
	RETURN;
END_IF

imageSizeInBytes := ULINT_TO_UDINT(imageInfo.nImageSize.Value);

IF imageSizeInBytes = 0 THEN
	TryDeserializeFrom := TRUE;
	RETURN;
END_IF

buffer := __NEW(BYTE, imageSizeInBytes);

IF NOT Deserializer.TryGetKeyBase64('imageData', buffer, imageSizeInBytes, Feedback) THEN
	__DELETE(buffer);
	RETURN;
END_IF

TryGetElementTypeFromInfo(imageInfo.Value, elementType);

hr := F_VN_CreateImageFromArray(
	pData := buffer,
	ipImage := activeData,
	nWidth := imageInfo.nWidth.Value,
	nHeight :=  imageInfo.nHeight.Value,
	ePixelType := elementType,
	nChannelNum := imageInfo.stPixelFormat.nChannels.Value, 
	hrPrev := hr);

__DELETE(buffer);

TryDeserializeFrom := TRUE;
END_METHOD

METHOD PUBLIC TryGetHeight : BOOL
VAR_INPUT
	Destination : REFERENCE TO UDINT;
END_VAR
IF NOT IsValid THEN
	RETURN;
END_IF

TryGetHeight := SUCCEEDED(activeData.GetHeight(Destination));
END_METHOD

METHOD PUBLIC TryGetImageData : BOOL
VAR_INPUT
	Destination : POINTER TO ITcVnData;
END_VAR
IF NOT IsValid THEN
	RETURN;
END_IF

TryGetImageData := SUCCEEDED(activeData.GetImageData(Destination));
END_METHOD

METHOD PUBLIC TryGetImageInfo : BOOL
VAR_INPUT
	Destination : REFERENCE TO  TcVnImageInfo;
END_VAR
IF NOT IsValid THEN
	RETURN;
END_IF

TryGetImageInfo := SUCCEEDED(activeData.GetImageInfo(Destination));
END_METHOD

METHOD PUBLIC TryGetImageSize : BOOL
VAR_INPUT
	Destination : REFERENCE TO ULINT;
END_VAR
IF NOT IsValid THEN
	RETURN;
END_IF

TryGetImageSize := SUCCEEDED(activeData.GetImageSize(Destination));
END_METHOD

METHOD PUBLIC TryGetPixelFormat : BOOL
VAR_INPUT
	Destination : REFERENCE TO  TcVnPixelFormat;
END_VAR
IF NOT IsValid THEN
	RETURN;
END_IF

TryGetPixelFormat := SUCCEEDED(activeData.GetPixelFormat(Destination));
END_METHOD

METHOD PUBLIC TryGetRowPointer : BOOL
VAR_INPUT
	RowIndex : UDINT;
	Destination : POINTER TO PVOID;
END_VAR
IF NOT IsValid THEN
	RETURN;
END_IF

TryGetRowPointer := SUCCEEDED(activeData.GetRowPointer(RowIndex, Destination));
END_METHOD

METHOD PUBLIC TryGetWidth : BOOL
VAR_INPUT
	Destination : REFERENCE TO UDINT;
END_VAR
IF NOT IsValid THEN
	RETURN;
END_IF

TryGetWidth := SUCCEEDED(activeData.GetWidth(Destination));
END_METHOD

METHOD PUBLIC TryGetXPadding : BOOL
VAR_INPUT
	Destination : REFERENCE TO UINT;
END_VAR
IF NOT IsValid THEN
	RETURN;
END_IF

TryGetXPadding := SUCCEEDED(activeData.GetXPadding(Destination));
END_METHOD

METHOD PUBLIC TryGetYPadding : BOOL
VAR_INPUT
	Destination : REFERENCE TO UINT;
END_VAR
IF NOT IsValid THEN
	RETURN;
END_IF

TryGetYPadding := SUCCEEDED(activeData.GetYPadding(Destination));
END_METHOD

METHOD PUBLIC TryReleaseRowPointer : BOOL
VAR_INPUT
	ppRow : POINTER TO PVOID;
END_VAR
IF NOT IsValid THEN
	RETURN;
END_IF

TryReleaseRowPointer := SUCCEEDED(activeData.ReleaseRowPointer(ppRow));
END_METHOD

METHOD PUBLIC TryTcAddRef : BOOL
VAR_INPUT
END_VAR
IF activeData = 0 THEN
	RETURN;
END_IF

IF activeData.TcAddRef() = 0 THEN
	activeData := 0;
END_IF

TryTcAddRef := TRUE;
END_METHOD

METHOD PUBLIC TryTcRelease : BOOL
VAR_INPUT
END_VAR
IF activeData = 0 THEN
	RETURN;
END_IF

IF activeData.TcRelease() = 0 THEN
	activeData := 0;
END_IF

TryTcRelease := TRUE;
END_METHOD

END_FUNCTION_BLOCK

// Datatypes/Structs/_TcVnImageInfo
{attribute 'linkalways'} 
{attribute 'no_explicit_call' := 'This FB is a CLASS and must be accessed using methods or properties'}
{attribute 'enable_dynamic_creation'}
FUNCTION_BLOCK _TcVnImageInfo EXTENDS StructuredDatatypeBase
VAR
	localData : TcVnImageInfo;
	activeData : REFERENCE TO TcVnImageInfo REF= localData;
	_nImageSize : _ULINT(localData.nImageSize);
	_nWidth : _UDINT(localData.nWidth);
	_nHeight : _UDINT(localData.nHeight);
	_nXPadding : _UINT(localData.nXPadding);
	_nYPadding : _UINT(localData.nYPadding);
	_stPixelFormat : _TcVnPixelFormat();
END_VAR

PROPERTY PUBLIC Address : PVOID
GET
Address := ADR(activeData);
END_GET
END_PROPERTY

METHOD PUBLIC ClearReference
VAR_INPUT
END_VAR
activeData REF= localData;
SetMemberReference();
END_METHOD

PROPERTY PUBLIC Size : UDINT
GET
Size := SIZEOF(activeData);
END_GET
END_PROPERTY

METHOD FB_init : BOOL
VAR_INPUT
	bInitRetains : BOOL; // if TRUE, the retain variables are initialized (warm start / cold start)
	bInCopyCode : BOOL;  // if TRUE, the instance afterwards gets moved into the copy code (online change)
END_VAR
SetMemberReference();
AddMember('nImageSize',_nImageSize);
AddMember('nWidth',_nWidth);
AddMember('nHeight',_nHeight);
AddMember('nXPadding',_nXPadding);
AddMember('nYPadding',_nYPadding);
AddMember('stPixelFormat',_stPixelFormat);
END_METHOD

METHOD PROTECTED SetMemberReference
VAR_INPUT
END_VAR
_nImageSize.MakeReferenceTo(activeData.nImageSize);
_nWidth.MakeReferenceTo(activeData.nWidth);
_nHeight.MakeReferenceTo(activeData.nHeight);
_nXPadding.MakeReferenceTo(activeData.nXPadding);
_nYPadding.MakeReferenceTo(activeData.nYPadding);
_stPixelFormat.MakeReferenceTo(activeData.stPixelFormat);
END_METHOD

METHOD PUBLIC Clone : I_Datatype
VAR
    pClone : POINTER TO _TcVnImageInfo;
END_VAR
pClone := __NEW(_TcVnImageInfo());
pClone^.Value := Value;
Clone := pClone^;
END_METHOD

PROPERTY PUBLIC Identifier : T_MAXSTRING
GET
Identifier := 'TcVnImageInfo';
END_GET
END_PROPERTY

METHOD PUBLIC MakeReferenceTo
VAR_INPUT
	ReferenceTarget : REFERENCE TO TcVnImageInfo;
END_VAR
activeData REF= ReferenceTarget;
SetMemberReference();
END_METHOD

METHOD TryMakeReferenceTo : BOOL
VAR_INPUT
	Target : I_Datatype;
END_VAR
VAR
	pTargetData : POINTER TO TcVnImageInfo;
END_VAR
IF NOT IsEquivalentTo(Target) THEN
	RETURN;
END_IF

pTargetData := Target.Address;
activeData REF= pTargetData^;
SetMemberReference();
TryMakeReferenceTo := TRUE;
END_METHOD

PROPERTY PUBLIC Value : reference to TcVnImageInfo
GET
Value ref= activeData;
END_GET
END_PROPERTY

PROPERTY PUBLIC nHeight : Reference to _UDINT
GET
nHeight REF= _nHeight;
END_GET
END_PROPERTY

PROPERTY PUBLIC nImageSize : Reference to _ULINT
GET
nImageSize REF= _nImageSize;
END_GET
END_PROPERTY

PROPERTY PUBLIC nWidth : Reference to _UDINT
GET
nWidth REF= _nWidth;
END_GET
END_PROPERTY

PROPERTY PUBLIC nXPadding : Reference to _UINT
GET
nXPadding REF= _nXPadding;
END_GET
END_PROPERTY

PROPERTY PUBLIC nYPadding : Reference to _UINT
GET
nYPadding REF= _nYPadding;
END_GET
END_PROPERTY

PROPERTY PUBLIC stPixelFormat : Reference to _TcVnPixelFormat
GET
stPixelFormat REF= _stPixelFormat;
END_GET
END_PROPERTY

END_FUNCTION_BLOCK

// Datatypes/Structs/_TcVnPixelFormat
{attribute 'linkalways'} 
{attribute 'no_explicit_call' := 'This FB is a CLASS and must be accessed using methods or properties'}
{attribute 'enable_dynamic_creation'}
FUNCTION_BLOCK _TcVnPixelFormat EXTENDS StructuredDatatypeBase
VAR
	localData : TcVnPixelFormat;
	activeData : REFERENCE TO TcVnPixelFormat REF= localData;

	_bSupported : _BIT();
	_bSigned : _BIT();
	_bPlanar : _BIT();
	_bFloat : _BIT();
	_nChannels : _BYTE(localData.nChannels);
	_ePixelEncoding : _ETcVnPixelEncoding(localData.ePixelEncoding);
	_ePixelPackMode : _ETcVnPixelPackMode(localData.ePixelPackMode);
	_nElementSize : _UINT(localData.nElementSize);
	_nTotalSize : _UINT(localData.nTotalSize);
END_VAR

PROPERTY PUBLIC Address : PVOID
GET
Address := ADR(activeData);
END_GET
END_PROPERTY

METHOD PUBLIC ClearReference
VAR_INPUT
END_VAR
activeData REF= localData;
SetMemberReference();
END_METHOD

PROPERTY PUBLIC Size : UDINT
GET
Size := SIZEOF(activeData);
END_GET
END_PROPERTY

METHOD FB_init : BOOL
VAR_INPUT
	bInitRetains : BOOL; // if TRUE, the retain variables are initialized (warm start / cold start)
	bInCopyCode : BOOL;  // if TRUE, the instance afterwards gets moved into the copy code (online change)
END_VAR
SetMemberReference();
AddMember('bSupported',_bSupported);
AddMember('bSigned',_bSigned);
AddMember('bPlanar',_bPlanar);
AddMember('bFloat',_bFloat);
AddMember('nChannels',_nChannels);
AddMember('ePixelEncoding',_ePixelEncoding);
AddMember('ePixelPackMode',_ePixelPackMode);
AddMember('nElementSize',_nElementSize);
AddMember('nTotalSize',_nTotalSize);
END_METHOD

METHOD PROTECTED SetMemberReference
VAR_STAT
	// this variable is used for BITADR as this function failes if used on a local variable.
	structure : TcVnPixelFormat;
END_VAR
_bSupported.MakeReferenceTo(THIS^, GetByteOffset(localData, localData.bSupported), BITADR(structure.bSupported));
_bSigned.MakeReferenceTo(THIS^, GetByteOffset(localData, localData.bSigned), BITADR(structure.bSigned));
_bPlanar.MakeReferenceTo(THIS^, GetByteOffset(localData, localData.bPlanar), BITADR(structure.bPlanar));
_bFloat.MakeReferenceTo(THIS^, GetByteOffset(localData, localData.bFloat), BITADR(structure.bFloat));
_nChannels.MakeReferenceTo(activeData.nChannels);
_ePixelEncoding.MakeReferenceTo(activeData.ePixelEncoding);
_ePixelPackMode.MakeReferenceTo(activeData.ePixelPackMode);
_nElementSize.MakeReferenceTo(activeData.nElementSize);
_nTotalSize.MakeReferenceTo(activeData.nTotalSize);
END_METHOD

METHOD PUBLIC Clone : I_Datatype
VAR
    pClone : POINTER TO _TcVnPixelFormat;
END_VAR
pClone := __NEW(_TcVnPixelFormat());
pClone^.Value := Value;
Clone := pClone^;
END_METHOD

PROPERTY PUBLIC Identifier : T_MAXSTRING
GET
Identifier := 'TcVnPixelFormat';
END_GET
END_PROPERTY

METHOD PUBLIC MakeReferenceTo
VAR_INPUT
	ReferenceTarget : REFERENCE TO TcVnPixelFormat;
END_VAR
activeData REF= ReferenceTarget;
SetMemberReference();
END_METHOD

METHOD TryMakeReferenceTo : BOOL
VAR_INPUT
	Target : I_Datatype;
END_VAR
VAR
	pTargetData : POINTER TO TcVnPixelFormat;
END_VAR
IF NOT IsEquivalentTo(Target) THEN
	RETURN;
END_IF

pTargetData := Target.Address;
activeData REF= pTargetData^;
SetMemberReference();
TryMakeReferenceTo := TRUE;
END_METHOD

PROPERTY PUBLIC Value : reference to TcVnPixelFormat
GET
Value REF= activeData;
END_GET
END_PROPERTY

PROPERTY PUBLIC bFloat : Reference to _BIT
GET
bFloat REF= _bFloat;
END_GET
END_PROPERTY

PROPERTY PUBLIC bPlanar : Reference to _BIT
GET
bPlanar REF= _bPlanar;
END_GET
END_PROPERTY

PROPERTY PUBLIC bSigned : Reference to _BIT
GET
bSigned REF= _bSigned;
END_GET
END_PROPERTY

PROPERTY PUBLIC bSupported : Reference to _BIT
GET
bSupported REF= _bSupported;
END_GET
END_PROPERTY

PROPERTY PUBLIC ePixelEncoding : Reference to _ETcVnPixelEncoding
GET
ePixelEncoding REF= _ePixelEncoding;
END_GET
END_PROPERTY

PROPERTY PUBLIC ePixelPackMode : Reference to _ETcVnPixelPackMode
GET
ePixelPackMode REF= _ePixelPackMode;
END_GET
END_PROPERTY

PROPERTY PUBLIC nChannels : Reference to _BYTE
GET
nChannels REF= _nChannels;
END_GET
END_PROPERTY

PROPERTY PUBLIC nElementSize : Reference to _UINT
GET
nElementSize REF= _nElementSize;
END_GET
END_PROPERTY

PROPERTY PUBLIC nTotalSize : Reference to _UINT
GET
nTotalSize REF= _nTotalSize;
END_GET
END_PROPERTY

END_FUNCTION_BLOCK

// Datatypes/Enums/_ETcVnPixelEncoding
{attribute 'linkalways'} 
{attribute 'no_explicit_call' := 'This FB is a CLASS and must be accessed using methods or properties'}
{attribute 'enable_dynamic_creation'}
FUNCTION_BLOCK _ETcVnPixelEncoding EXTENDS EnumDatatypeBase
VAR
	localData : ETcVnPixelEncoding;
	activeData : REFERENCE TO ETcVnPixelEncoding;
	enumBaseDatatype : _BYTE(localData);
END_VAR

METHOD PROTECTED SetBaseDatatypeReference
VAR_INPUT
END_VAR
enumBaseDatatype.MakeReferenceTo(activeData);
END_METHOD

PROPERTY PUBLIC Address : PVOID
GET
Address := ADR(activeData);
END_GET
END_PROPERTY

METHOD PUBLIC ClearReference
VAR_INPUT
END_VAR
activeData REF= localData;
SetBaseDatatypeReference();
END_METHOD

PROPERTY PUBLIC Size : UDINT
GET
Size := SIZEOF(activeData);
END_GET
END_PROPERTY

METHOD FB_init : BOOL
VAR_INPUT
	bInitRetains : BOOL; // if TRUE, the retain variables are initialized (warm start / cold start)
	bInCopyCode : BOOL;  // if TRUE, the instance afterwards gets moved into the copy code (online change)
	InitialValue : ETcVnPixelEncoding;
END_VAR
localData := InitialValue;
AddBaseDatatype(enumBaseDatatype);
ClearReference();

AddLocalEnumeration('TCVN_PE_NONE', ETcVnPixelEncoding.TCVN_PE_NONE);
AddLocalEnumeration('TCVN_PE_BAYER_GR', ETcVnPixelEncoding.TCVN_PE_BAYER_GR);
AddLocalEnumeration('TCVN_PE_BAYER_RG', ETcVnPixelEncoding.TCVN_PE_BAYER_RG);
AddLocalEnumeration('TCVN_PE_BAYER_GB', ETcVnPixelEncoding.TCVN_PE_BAYER_GB);
AddLocalEnumeration('TCVN_PE_BAYER_BG', ETcVnPixelEncoding.TCVN_PE_BAYER_BG);
AddLocalEnumeration('TCVN_PE_YUV_411_UYYVYY', ETcVnPixelEncoding.TCVN_PE_YUV_411_UYYVYY);
AddLocalEnumeration('TCVN_PE_YUV_422_UYVY', ETcVnPixelEncoding.TCVN_PE_YUV_422_UYVY);
AddLocalEnumeration('TCVN_PE_YUV_422_YUYV', ETcVnPixelEncoding.TCVN_PE_YUV_422_YUYV);
AddLocalEnumeration('TCVN_PE_YCBCR_411_CBYYCRYY', ETcVnPixelEncoding.TCVN_PE_YCBCR_411_CBYYCRYY);
AddLocalEnumeration('TCVN_PE_YCBCR_422_CBYCRY', ETcVnPixelEncoding.TCVN_PE_YCBCR_422_CBYCRY);
AddLocalEnumeration('TCVN_PE_YCBCR_422_YCBYCR', ETcVnPixelEncoding.TCVN_PE_YCBCR_422_YCBYCR);
END_METHOD

METHOD PRIVATE AddLocalEnumeration
VAR_INPUT
	Enumeration : T_MAXSTRING;
	Value : ETcVnPixelEncoding;
END_VAR
AddEnumeration(Enumeration, Value);
END_METHOD

METHOD IsEnumeratorValueEqual : BOOL
VAR_INPUT
	Enumerator : I_KeyValueForwardEnumerator;
END_VAR
VAR
	storedValue : ETcVnPixelEncoding;
END_VAR
IF NOT Enumerator.TryGet(storedValue) THEN
	RETURN;
END_IF

IsEnumeratorValueEqual := storedValue = activeData;
END_METHOD

METHOD PUBLIC Clone : I_Datatype
VAR
    pClone : POINTER TO _ETcVnPixelEncoding;
END_VAR
pClone := __NEW(_ETcVnPixelEncoding(InitialValue := Value));
Clone := pClone^;
END_METHOD

PROPERTY PUBLIC Identifier : T_MAXSTRING
GET
Identifier := 'ETcVnPixelEncoding';
END_GET
END_PROPERTY

METHOD PUBLIC MakeReferenceTo
VAR_INPUT
	ReferenceTarget : REFERENCE TO ETcVnPixelEncoding;
END_VAR
activeData REF= ReferenceTarget;
SetBaseDatatypeReference();
END_METHOD

METHOD TryMakeReferenceTo : BOOL
VAR_INPUT
	Target : I_Datatype;
END_VAR
VAR
	pTargetData : POINTER TO ETcVnPixelEncoding;
END_VAR
IF NOT IsEquivalentTo(Target) THEN
	RETURN;
END_IF

pTargetData := Target.Address;
activeData REF= pTargetData^;
SetBaseDatatypeReference();
TryMakeReferenceTo := TRUE;
END_METHOD

PROPERTY PUBLIC Value : ETcVnPixelEncoding
GET
Value := activeData;
END_GET
SET
activeData := Value;
END_SET
END_PROPERTY

END_FUNCTION_BLOCK

// Datatypes/Enums/_ETcVnPixelPackMode
{attribute 'linkalways'} 
{attribute 'no_explicit_call' := 'This FB is a CLASS and must be accessed using methods or properties'}
{attribute 'enable_dynamic_creation'}
FUNCTION_BLOCK _ETcVnPixelPackMode EXTENDS EnumDatatypeBase
VAR
	localData : ETcVnPixelPackMode;
	activeData : REFERENCE TO ETcVnPixelPackMode;
	enumBaseDatatype : _BYTE(localData);
END_VAR

METHOD PROTECTED SetBaseDatatypeReference
VAR_INPUT
END_VAR
enumBaseDatatype.MakeReferenceTo(activeData);
END_METHOD

PROPERTY PUBLIC Address : PVOID
GET
Address := ADR(activeData);
END_GET
END_PROPERTY

METHOD PUBLIC ClearReference
VAR_INPUT
END_VAR
activeData REF= localData;
SetBaseDatatypeReference();
END_METHOD

PROPERTY PUBLIC Size : UDINT
GET
Size := SIZEOF(activeData);
END_GET
END_PROPERTY

METHOD FB_init : BOOL
VAR_INPUT
	bInitRetains : BOOL; // if TRUE, the retain variables are initialized (warm start / cold start)
	bInCopyCode : BOOL;  // if TRUE, the instance afterwards gets moved into the copy code (online change)
	InitialValue : ETcVnPixelPackMode;
END_VAR
localData := InitialValue;
AddBaseDatatype(enumBaseDatatype);
ClearReference();

AddLocalEnumeration('TCVN_PPM_NONE', ETcVnPixelPackMode.TCVN_PPM_NONE);
AddLocalEnumeration('TCVN_PPM_MONO1P', ETcVnPixelPackMode.TCVN_PPM_MONO1P);
AddLocalEnumeration('TCVN_PPM_MONO2P', ETcVnPixelPackMode.TCVN_PPM_MONO2P);
AddLocalEnumeration('TCVN_PPM_MONO4P', ETcVnPixelPackMode.TCVN_PPM_MONO4P);
AddLocalEnumeration('TCVN_PPM_MONO10PACKED', ETcVnPixelPackMode.TCVN_PPM_MONO10PACKED);
AddLocalEnumeration('TCVN_PPM_MONO12PACKED', ETcVnPixelPackMode.TCVN_PPM_MONO12PACKED);
AddLocalEnumeration('TCVN_PPM_RGB10V1PACKED', ETcVnPixelPackMode.TCVN_PPM_RGB10V1PACKED);
AddLocalEnumeration('TCVN_PPM_RGB10P32', ETcVnPixelPackMode.TCVN_PPM_RGB10P32);
AddLocalEnumeration('TCVN_PPM_RGB12V1PACKED', ETcVnPixelPackMode.TCVN_PPM_RGB12V1PACKED);
AddLocalEnumeration('TCVN_PPM_RGB565P', ETcVnPixelPackMode.TCVN_PPM_RGB565P);
AddLocalEnumeration('TCVN_PPM_BGR565P', ETcVnPixelPackMode.TCVN_PPM_BGR565P);
AddLocalEnumeration('TCVN_PPM_MONO10P', ETcVnPixelPackMode.TCVN_PPM_MONO10P);
AddLocalEnumeration('TCVN_PPM_MONO12P', ETcVnPixelPackMode.TCVN_PPM_MONO12P);
END_METHOD

METHOD PRIVATE AddLocalEnumeration
VAR_INPUT
	Enumeration : T_MAXSTRING;
	Value : ETcVnPixelPackMode;
END_VAR
AddEnumeration(Enumeration, Value);
END_METHOD

METHOD IsEnumeratorValueEqual : BOOL
VAR_INPUT
	Enumerator : I_KeyValueForwardEnumerator;
END_VAR
VAR
	storedValue : ETcVnPixelPackMode;
END_VAR
IF NOT Enumerator.TryGet(storedValue) THEN
	RETURN;
END_IF

IsEnumeratorValueEqual := storedValue = activeData;
END_METHOD

METHOD PUBLIC Clone : I_Datatype
VAR
    pClone : POINTER TO _ETcVnPixelPackMode;
END_VAR
pClone := __NEW(_ETcVnPixelPackMode(InitialValue := Value));
Clone := pClone^;
END_METHOD

PROPERTY PUBLIC Identifier : T_MAXSTRING
GET
Identifier := 'ETcVnPixelPackMode';
END_GET
END_PROPERTY

METHOD PUBLIC MakeReferenceTo
VAR_INPUT
	ReferenceTarget : REFERENCE TO ETcVnPixelPackMode;
END_VAR
activeData REF= ReferenceTarget;
SetBaseDatatypeReference();
END_METHOD

METHOD TryMakeReferenceTo : BOOL
VAR_INPUT
	Target : I_Datatype;
END_VAR
VAR
	pTargetData : POINTER TO ETcVnPixelPackMode;
END_VAR
IF NOT IsEquivalentTo(Target) THEN
	RETURN;
END_IF

pTargetData := Target.Address;
activeData REF= pTargetData^;
SetBaseDatatypeReference();
TryMakeReferenceTo := TRUE;
END_METHOD

PROPERTY PUBLIC Value : ETcVnPixelPackMode
GET
Value := activeData;
END_GET
SET
activeData := Value;
END_SET
END_PROPERTY

END_FUNCTION_BLOCK

// Datatypes/Aliases/_TcVnArray3_Point2_REAL
{attribute 'linkalways'} 
{attribute 'no_explicit_call' := 'This FB is a CLASS and must be accessed using methods or properties'}
{attribute 'enable_dynamic_creation'}
FUNCTION_BLOCK _TcVnArray3_Point2_REAL EXTENDS AliasDatatypeBase
VAR
	localData : TcVnArray3_Point2_REAL;
	activeData : REFERENCE TO TcVnArray3_Point2_REAL REF= localData;
	aliasBaseDatatype : _Array0to2OfTcVnPoint2_REAL;
END_VAR

METHOD PROTECTED SetBaseDatatypeReference
VAR_INPUT
END_VAR
aliasBaseDatatype.MakeReferenceTo(activeData);
END_METHOD

PROPERTY PUBLIC Address : PVOID
GET
Address := ADR(activeData);
END_GET
END_PROPERTY

METHOD PUBLIC ClearReference
VAR_INPUT
END_VAR
activeData REF= localData;
SetBaseDatatypeReference();
END_METHOD

PROPERTY PUBLIC Size : UDINT
GET
Size := SIZEOF(activeData);
END_GET
END_PROPERTY

METHOD FB_init : BOOL
VAR_INPUT
	bInitRetains : BOOL; // if TRUE, the retain variables are initialized (warm start / cold start)
	bInCopyCode : BOOL;  // if TRUE, the instance afterwards gets moved into the copy code (online change)
	//InitialValue : TcVnArray4_LREAL; // if possible, not all values can be initialized
END_VAR
//localData := InitialValue; // if possible, not all values can be initialized
SetBaseDatatypeReference();
AddBaseDatatype(aliasBaseDatatype);
END_METHOD

METHOD PUBLIC Clone : I_Datatype
VAR
    pClone : POINTER TO _TcVnArray3_Point2_REAL;
END_VAR
pClone := __NEW(_TcVnArray3_Point2_REAL);
Clone := pClone^;
END_METHOD

PROPERTY PUBLIC Identifier : T_MAXSTRING
GET
Identifier := 'TcVnArray3_Point2_REAL';
END_GET
END_PROPERTY

METHOD PUBLIC MakeReferenceTo
VAR_INPUT
	ReferenceTarget : REFERENCE TO TcVnArray3_Point2_REAL;
END_VAR
activeData REF= ReferenceTarget;
SetBaseDatatypeReference();
END_METHOD

METHOD TryMakeReferenceTo : BOOL
VAR_INPUT
	Target : I_Datatype;
END_VAR
VAR
	pTargetData : POINTER TO TcVnArray3_Point2_REAL;
END_VAR
IF NOT IsEquivalentTo(Target) THEN
	RETURN;
END_IF

pTargetData := Target.Address;
activeData REF= pTargetData^;
SetBaseDatatypeReference();
TryMakeReferenceTo := TRUE;
END_METHOD

PROPERTY PUBLIC Value : REFERENCE TO TcVnArray3_Point2_REAL
GET
Value REF= activeData;
END_GET
END_PROPERTY

END_FUNCTION_BLOCK

// Datatypes/Arrays/_Array0to2OfTcVnPoint2_REAL
{attribute 'linkalways'} 
{attribute 'no_explicit_call' := 'This FB is a CLASS and must be accessed using methods or properties'}
{attribute 'enable_dynamic_creation'}
FUNCTION_BLOCK _Array0to2OfTcVnPoint2_REAL EXTENDS ArrayDatatypeBase_1D
VAR CONSTANT
	lBound : DINT := 0;
	uBound : DINT := 2;
END_VAR
VAR
	localData : ARRAY [lBound..uBound] OF TcVnPoint2_REAL;
	activeData : REFERENCE TO ARRAY [lBound..uBound] OF TcVnPoint2_REAL REF= localData;
	elements : ARRAY [lBound..uBound] OF _TcVnPoint2_REAL;
	baseType : _TcVnPoint2_REAL;
END_VAR

METHOD FB_init : BOOL
VAR_INPUT
	bInitRetains : BOOL; // if TRUE, the retain variables are initialized (warm start / cold start)
	bInCopyCode : BOOL;  // if TRUE, the instance afterwards gets moved into the copy code (online change)
END_VAR
SetElementReference();
END_METHOD

METHOD PROTECTED OnSerializeArrayValues
VAR_INPUT
	Serializer : I_Serializer;
END_VAR
VAR
	i : DINT;
END_VAR
FOR i := lBound TO uBound DO
	elements[i].SerializeWith(Serializer);
END_FOR
END_METHOD

METHOD PROTECTED SetElementReference
VAR_INPUT
END_VAR
VAR
	i : DINT;
END_VAR
FOR i := lBound TO uBound DO
	elements[i].MakeReferenceTo(activeData[i]);
END_FOR
END_METHOD

METHOD PROTECTED TryDeserializeArrayValues : BOOL
VAR_INPUT
	Deserializer : I_Deserializer;
	Feedback : I_DeserializerFeedback;
END_VAR
VAR
	enumerator : I_DeserializerArrayForwardEnumerator;
	i : DINT;
END_VAR
enumerator := Deserializer.GetArrayEnumerator();
i := lBound;

WHILE enumerator.MoveNext() AND i <= uBound DO
	
	IF NOT elements[i].TryDeserializeFrom(enumerator.Current, Feedback) THEN
		EXIT;
	END_IF
	i := i + 1;

END_WHILE
enumerator.Dispose();
END_METHOD

PROPERTY PUBLIC Address : PVOID
GET
Address := ADR(activeData);
END_GET
END_PROPERTY

PROPERTY PUBLIC BaseDatatype : I_Datatype
GET
BaseDatatype := baseType;
END_GET
END_PROPERTY

METHOD PUBLIC ClearReference
VAR_INPUT
END_VAR
activeData REF= localData;
SetElementReference();
END_METHOD

PROPERTY PUBLIC Size : UDINT
GET
Size := SIZEOF(activeData);
END_GET
END_PROPERTY

METHOD PUBLIC TryGetElementAsDatatypeByIndex : BOOL
VAR_INPUT
	Index : DINT;
	Destination : REFERENCE TO I_Datatype;
END_VAR
IF Index < lbound OR Index > ubound THEN
	RETURN;
END_IF

Destination := elements[Index];
TryGetElementAsDatatypeByIndex := TRUE;
END_METHOD

METHOD PUBLIC TryGetLowerBound : BOOL
VAR_INPUT
	Dimention : UDINT;
	Destination : REFERENCE TO DINT;
END_VAR
IF Dimention = 1 THEN
	Destination := lBound;
	TryGetLowerBound := TRUE;
END_IF
END_METHOD

METHOD PUBLIC TryGetUpperBound : BOOL
VAR_INPUT
	Dimention : UDINT;
	Destination : REFERENCE TO DINT;
END_VAR
IF Dimention = 1 THEN
	Destination := uBound;
	TryGetUpperBound := TRUE;
END_IF
END_METHOD

METHOD PUBLIC Clone : I_Datatype
VAR
    pClone : POINTER TO _Array0to2OfTcVnPoint2_REAL;
END_VAR
pClone := __NEW(_Array0to2OfTcVnPoint2_REAL());
pClone^.Value := Value;
Clone := pClone^;
END_METHOD

METHOD PUBLIC MakeReferenceTo
VAR_INPUT
	ReferenceTarget : REFERENCE TO ARRAY [lBound..uBound] OF TcVnPoint2_REAL;
END_VAR
activeData REF= ReferenceTarget;
SetElementReference();
END_METHOD

METHOD TryMakeReferenceTo : BOOL
VAR_INPUT
	Target : I_Datatype;
END_VAR
VAR
	pTargetData : POINTER TO ARRAY [lBound..uBound] OF TcVnPoint2_REAL;
END_VAR
IF NOT IsEquivalentTo(Target) THEN
	RETURN;
END_IF

pTargetData := Target.Address;
activeData REF= pTargetData^;
SetElementReference();
TryMakeReferenceTo := TRUE;
END_METHOD

PROPERTY PUBLIC Value : REFERENCE TO ARRAY [lBound..uBound] OF TcVnPoint2_REAL;
GET
Value ref= activeData;
END_GET
END_PROPERTY

END_FUNCTION_BLOCK

// Datatypes/Aliases/_TcVnPoint2_REAL
{attribute 'linkalways'} 
{attribute 'no_explicit_call' := 'This FB is a CLASS and must be accessed using methods or properties'}
{attribute 'enable_dynamic_creation'}
FUNCTION_BLOCK _TcVnPoint2_REAL EXTENDS AliasDatatypeBase
VAR
	localData : TcVnPoint2_REAL;
	activeData : REFERENCE TO TcVnPoint2_REAL REF= localData;
	aliasBaseDatatype : _TcVnVector2_REAL;
END_VAR

METHOD PROTECTED SetBaseDatatypeReference
VAR_INPUT
END_VAR
aliasBaseDatatype.MakeReferenceTo(activeData);
END_METHOD

PROPERTY PUBLIC Address : PVOID
GET
Address := ADR(activeData);
END_GET
END_PROPERTY

METHOD PUBLIC ClearReference
VAR_INPUT
END_VAR
activeData REF= localData;
SetBaseDatatypeReference();
END_METHOD

PROPERTY PUBLIC Size : UDINT
GET
Size := SIZEOF(activeData);
END_GET
END_PROPERTY

METHOD FB_init : BOOL
VAR_INPUT
	bInitRetains : BOOL; // if TRUE, the retain variables are initialized (warm start / cold start)
	bInCopyCode : BOOL;  // if TRUE, the instance afterwards gets moved into the copy code (online change)
	//InitialValue : <type>; // if possible, not all values can be initialized
END_VAR
//localData := InitialValue; // if possible, not all values can be initialized
SetBaseDatatypeReference();
AddBaseDatatype(aliasBaseDatatype);
END_METHOD

